ABB RAPID module: P103.mod

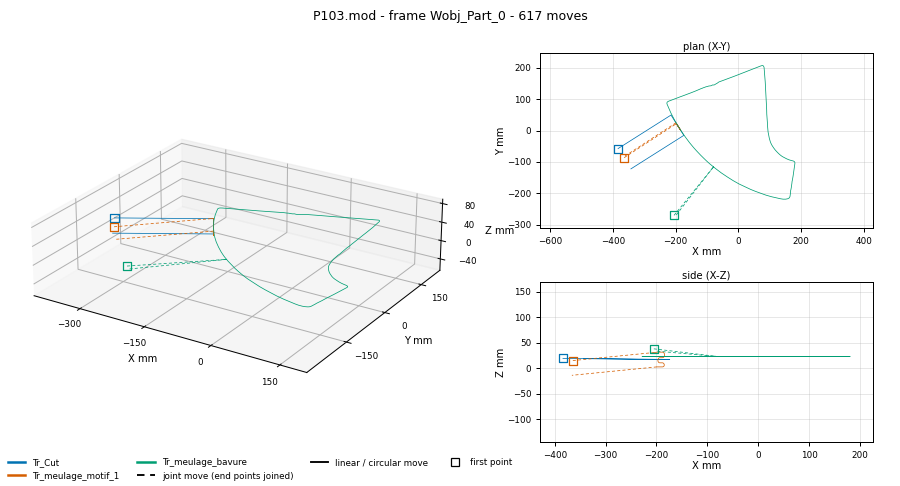
[picture p0: tool path of P103.mod in frame Wobj_Part_0, 617 of 625 moves have a stored position in this frame; points joined in program order, loops and branches not executed]
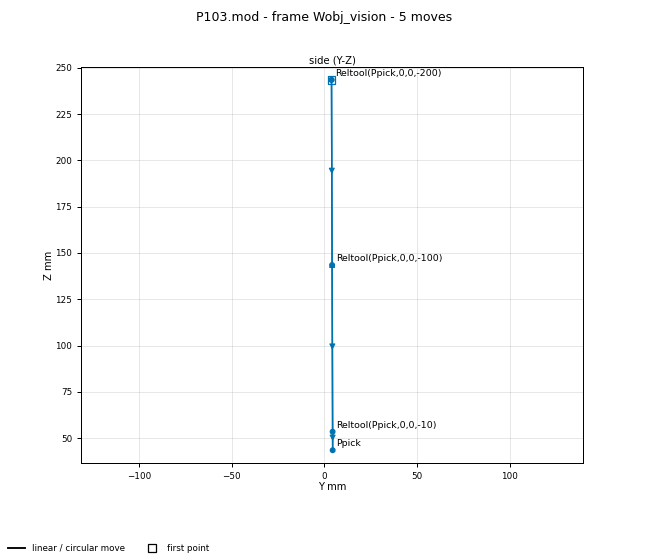
[picture p1: tool path of P103.mod in frame Wobj_vision, 5 of 625 moves have a stored position in this frame; points joined in program order, loops and branches not executed]
MODULE P103
	LOCAL CONST Speeddata vitesse_Tronconnage :=[10, 500, 0, 0];
	LOCAL CONST Robtarget Coupe_0 :=[[-191.77609375,12.892310546875,17.173708984375],[0.680249271326253,0.678001155670585,0.200784543502111,0.193030901308835],[0,0,0,0],[8.999999E+09,8.999999E+09,8.999999E+09,8.999999E+09,8.999999E+09,8.999999E+09]];
	LOCAL CONST Robtarget Tr_meulage_motif_1_App1 :=[[-364.480910820686,-86.5896332823026,15.1430730099713],[0.64692434542493,-0.59549439899172,0.32258675367408,-0.350446998018296],[0,0,0,0],[8.999999E+09,8.999999E+09,8.999999E+09,8.999999E+09,8.999999E+09,8.999999E+09]];
	LOCAL CONST Robtarget Tr_meulage_motif_1_App2 :=[[-205.877100228534,16.8426673593224,30.8462717169048],[0.64692434542493,-0.59549439899172,0.32258675367408,-0.350446998018296],[0,0,0,0],[8.999999E+09,8.999999E+09,8.999999E+09,8.999999E+09,8.999999E+09,8.999999E+09]];
	LOCAL CONST Robtarget Tr_meulage_motif_1_P0 :=[[-197.52953125,22.28647265625,31.672755859375],[0.64692434542493,-0.59549439899172,0.32258675367408,-0.350446998018296],[0,0,0,0],[8.999999E+09,8.999999E+09,8.999999E+09,8.999999E+09,8.999999E+09,8.999999E+09]];
	LOCAL CONST Robtarget Tr_meulage_motif_1_P1 :=[[-196.9945,21.441646484375,31.672755859375],[0.64692434542493,-0.59549439899172,0.32258675367408,-0.350446998018296],[0,0,0,0],[8.999999E+09,8.999999E+09,8.999999E+09,8.999999E+09,8.999999E+09,8.999999E+09]];
	LOCAL CONST Robtarget Tr_meulage_motif_1_P2 :=[[-196.459453125,20.5968203125,31.6727578125],[0.64692434542493,-0.59549439899172,0.32258675367408,-0.350446998018296],[0,0,0,0],[8.999999E+09,8.999999E+09,8.999999E+09,8.999999E+09,8.999999E+09,8.999999E+09]];
	LOCAL CONST Robtarget Tr_meulage_motif_1_P3 :=[[-195.92440625,19.75199609375,31.6727578125],[0.64692434542493,-0.59549439899172,0.32258675367408,-0.350446998018296],[0,0,0,0],[8.999999E+09,8.999999E+09,8.999999E+09,8.999999E+09,8.999999E+09,8.999999E+09]];
	LOCAL CONST Robtarget Tr_meulage_motif_1_P4 :=[[-195.389375,18.907169921875,31.6727578125],[0.64692434542493,-0.59549439899172,0.32258675367408,-0.350446998018296],[0,0,0,0],[8.999999E+09,8.999999E+09,8.999999E+09,8.999999E+09,8.999999E+09,8.999999E+09]];
	LOCAL CONST Robtarget Tr_meulage_motif_1_P5 :=[[-194.854328125,18.06234375,31.672759765625],[0.64692434542493,-0.59549439899172,0.32258675367408,-0.350446998018296],[0,0,0,0],[8.999999E+09,8.999999E+09,8.999999E+09,8.999999E+09,8.999999E+09,8.999999E+09]];
	LOCAL CONST Robtarget Tr_meulage_motif_1_P6 :=[[-194.31928125,17.217517578125,31.672759765625],[0.64692434542493,-0.59549439899172,0.32258675367408,-0.350446998018296],[0,0,0,0],[8.999999E+09,8.999999E+09,8.999999E+09,8.999999E+09,8.999999E+09,8.999999E+09]];
	LOCAL CONST Robtarget Tr_meulage_motif_1_P7 :=[[-193.78425,16.3726923828125,31.672759765625],[0.64692434542493,-0.59549439899172,0.32258675367408,-0.350446998018296],[0,0,0,0],[8.999999E+09,8.999999E+09,8.999999E+09,8.999999E+09,8.999999E+09,8.999999E+09]];
	LOCAL CONST Robtarget Tr_meulage_motif_1_P8 :=[[-193.249203125,15.5278671875,31.67276171875],[0.64692434542493,-0.59549439899172,0.32258675367408,-0.350446998018296],[0,0,0,0],[8.999999E+09,8.999999E+09,8.999999E+09,8.999999E+09,8.999999E+09,8.999999E+09]];
	LOCAL CONST Robtarget Tr_meulage_motif_1_P9 :=[[-192.71415625,14.683041015625,31.67276171875],[0.64692434542493,-0.59549439899172,0.32258675367408,-0.350446998018296],[0,0,0,0],[8.999999E+09,8.999999E+09,8.999999E+09,8.999999E+09,8.999999E+09,8.999999E+09]];
	LOCAL CONST Robtarget Tr_meulage_motif_1_P10 :=[[-192.179125,13.8382158203125,31.67276171875],[0.64692434542493,-0.59549439899172,0.32258675367408,-0.350446998018296],[0,0,0,0],[8.999999E+09,8.999999E+09,8.999999E+09,8.999999E+09,8.999999E+09,8.999999E+09]];
	LOCAL CONST Robtarget Tr_meulage_motif_1_P11 :=[[-191.644078125,12.9933896484375,31.672763671875],[0.64692434542493,-0.59549439899172,0.32258675367408,-0.350446998018296],[0,0,0,0],[8.999999E+09,8.999999E+09,8.999999E+09,8.999999E+09,8.999999E+09,8.999999E+09]];
	LOCAL CONST Robtarget Tr_meulage_motif_1_P12 :=[[-191.10903125,12.148564453125,31.672763671875],[0.64692434542493,-0.59549439899172,0.32258675367408,-0.350446998018296],[0,0,0,0],[8.999999E+09,8.999999E+09,8.999999E+09,8.999999E+09,8.999999E+09,8.999999E+09]];
	LOCAL CONST Robtarget Tr_meulage_motif_1_P13 :=[[-190.574,11.30373828125,31.672763671875],[0.64692434542493,-0.59549439899172,0.32258675367408,-0.350446998018296],[0,0,0,0],[8.999999E+09,8.999999E+09,8.999999E+09,8.999999E+09,8.999999E+09,8.999999E+09]];
	LOCAL CONST Robtarget Tr_meulage_motif_1_P14 :=[[-190.038953125,10.4589130859375,31.672765625],[0.64692434542493,-0.59549439899172,0.32258675367408,-0.350446998018296],[0,0,0,0],[8.999999E+09,8.999999E+09,8.999999E+09,8.999999E+09,8.999999E+09,8.999999E+09]];
	LOCAL CONST Robtarget Tr_meulage_motif_1_P15 :=[[-189.50390625,9.6140869140625,31.672765625],[0.64692434542493,-0.59549439899172,0.32258675367408,-0.350446998018296],[0,0,0,0],[8.999999E+09,8.999999E+09,8.999999E+09,8.999999E+09,8.999999E+09,8.999999E+09]];
	LOCAL CONST Robtarget Tr_meulage_motif_1_P16 :=[[-188.968875,8.76926171875,31.672765625],[0.64692434542493,-0.59549439899172,0.32258675367408,-0.350446998018296],[0,0,0,0],[8.999999E+09,8.999999E+09,8.999999E+09,8.999999E+09,8.999999E+09,8.999999E+09]];
	LOCAL CONST Robtarget Tr_meulage_motif_1_P17 :=[[-188.433828125,7.92443603515625,31.672767578125],[0.64692434542493,-0.59549439899172,0.32258675367408,-0.350446998018296],[0,0,0,0],[8.999999E+09,8.999999E+09,8.999999E+09,8.999999E+09,8.999999E+09,8.999999E+09]];
	LOCAL CONST Robtarget Tr_meulage_motif_1_P18 :=[[-187.89878125,7.0796103515625,31.672767578125],[0.64692434542493,-0.59549439899172,0.32258675367408,-0.350446998018296],[0,0,0,0],[8.999999E+09,8.999999E+09,8.999999E+09,8.999999E+09,8.999999E+09,8.999999E+09]];
	LOCAL CONST Robtarget Tr_meulage_motif_1_P19 :=[[-187.368796875,6.24039208984375,31.562181640625],[0.64692434542493,-0.59549439899172,0.32258675367408,-0.350446998018296],[0,0,0,0],[8.999999E+09,8.999999E+09,8.999999E+09,8.999999E+09,8.999999E+09,8.999999E+09]];
	LOCAL CONST Robtarget Tr_meulage_motif_1_P20 :=[[-186.86440625,5.4394736328125,31.351009765625],[0.64692434542493,-0.59549439899172,0.32258675367408,-0.350446998018296],[0,0,0,0],[8.999999E+09,8.999999E+09,8.999999E+09,8.999999E+09,8.999999E+09,8.999999E+09]];
	LOCAL CONST Robtarget Tr_meulage_motif_1_P21 :=[[-186.410796875,4.71741357421875,31.07918359375],[0.64692434542493,-0.59549439899172,0.32258675367408,-0.350446998018296],[0,0,0,0],[8.999999E+09,8.999999E+09,8.999999E+09,8.999999E+09,8.999999E+09,8.999999E+09]];
	LOCAL CONST Robtarget Tr_meulage_motif_1_P22 :=[[-186.012203125,4.08216088867187,30.803263671875],[0.64692434542493,-0.59549439899172,0.32258675367408,-0.350446998018296],[0,0,0,0],[8.999999E+09,8.999999E+09,8.999999E+09,8.999999E+09,8.999999E+09,8.999999E+09]];
	LOCAL CONST Robtarget Tr_meulage_motif_1_P23 :=[[-185.42903125,3.148189453125,30.1871796875],[0.64692434542493,-0.59549439899172,0.32258675367408,-0.350446998018296],[0,0,0,0],[8.999999E+09,8.999999E+09,8.999999E+09,8.999999E+09,8.999999E+09,8.999999E+09]];
	LOCAL CONST Robtarget Tr_meulage_motif_1_P24 :=[[-184.88940625,2.27801293945312,29.339580078125],[0.64692434542493,-0.59549439899172,0.32258675367408,-0.350446998018296],[0,0,0,0],[8.999999E+09,8.999999E+09,8.999999E+09,8.999999E+09,8.999999E+09,8.999999E+09]];
	LOCAL CONST Robtarget Tr_meulage_motif_1_P25 :=[[-184.44575,1.55563366699219,28.315771484375],[0.64692434542493,-0.59549439899172,0.32258675367408,-0.350446998018296],[0,0,0,0],[8.999999E+09,8.999999E+09,8.999999E+09,8.999999E+09,8.999999E+09,8.999999E+09]];
	LOCAL CONST Robtarget Tr_meulage_motif_1_P26 :=[[-184.195328125,1.13640502929688,27.199658203125],[0.64692434542493,-0.59549439899172,0.32258675367408,-0.350446998018296],[0,0,0,0],[8.999999E+09,8.999999E+09,8.999999E+09,8.999999E+09,8.999999E+09,8.999999E+09]];
	LOCAL CONST Robtarget Tr_meulage_motif_1_P27 :=[[-184.187578125,1.10928845214844,26.503734375],[0.64692434542493,-0.59549439899172,0.32258675367408,-0.350446998018296],[0,0,0,0],[8.999999E+09,8.999999E+09,8.999999E+09,8.999999E+09,8.999999E+09,8.999999E+09]];
	LOCAL CONST Robtarget Tr_meulage_motif_1_P28 :=[[-184.193953125,1.10524719238281,25.84252734375],[0.64692434542493,-0.59549439899172,0.32258675367408,-0.350446998018296],[0,0,0,0],[8.999999E+09,8.999999E+09,8.999999E+09,8.999999E+09,8.999999E+09,8.999999E+09]];
	LOCAL CONST Robtarget Tr_meulage_motif_1_P29 :=[[-184.2296875,1.14756665039062,25.1814765625],[0.64692434542493,-0.59549439899172,0.32258675367408,-0.350446998018296],[0,0,0,0],[8.999999E+09,8.999999E+09,8.999999E+09,8.999999E+09,8.999999E+09,8.999999E+09]];
	LOCAL CONST Robtarget Tr_meulage_motif_1_P30 :=[[-184.506890625,1.5617412109375,24.079798828125],[0.64692434542493,-0.59549439899172,0.32258675367408,-0.350446998018296],[0,0,0,0],[8.999999E+09,8.999999E+09,8.999999E+09,8.999999E+09,8.999999E+09,8.999999E+09]];
	LOCAL CONST Robtarget Tr_meulage_motif_1_P31 :=[[-184.9749375,2.27928784179687,23.07323828125],[0.64692434542493,-0.59549439899172,0.32258675367408,-0.350446998018296],[0,0,0,0],[8.999999E+09,8.999999E+09,8.999999E+09,8.999999E+09,8.999999E+09,8.999999E+09]];
	LOCAL CONST Robtarget Tr_meulage_motif_1_P32 :=[[-185.5305,3.13882202148437,22.24441796875],[0.64692434542493,-0.59549439899172,0.32258675367408,-0.350446998018296],[0,0,0,0],[8.999999E+09,8.999999E+09,8.999999E+09,8.999999E+09,8.999999E+09,8.999999E+09]];
	LOCAL CONST Robtarget Tr_meulage_motif_1_P33 :=[[-185.9019375,3.71687768554688,21.848693359375],[0.64692434542493,-0.59549439899172,0.32258675367408,-0.350446998018296],[0,0,0,0],[8.999999E+09,8.999999E+09,8.999999E+09,8.999999E+09,8.999999E+09,8.999999E+09]];
	LOCAL CONST Robtarget Tr_meulage_motif_1_P34 :=[[-186.526296875,4.69233837890625,21.36119140625],[0.64692434542493,-0.59549439899172,0.32258675367408,-0.350446998018296],[0,0,0,0],[8.999999E+09,8.999999E+09,8.999999E+09,8.999999E+09,8.999999E+09,8.999999E+09]];
	LOCAL CONST Robtarget Tr_meulage_motif_1_P35 :=[[-186.980984375,5.40462841796875,21.097115234375],[0.64692434542493,-0.59549439899172,0.32258675367408,-0.350446998018296],[0,0,0,0],[8.999999E+09,8.999999E+09,8.999999E+09,8.999999E+09,8.999999E+09,8.999999E+09]];
	LOCAL CONST Robtarget Tr_meulage_motif_1_P36 :=[[-187.481609375,6.19075634765625,20.89266015625],[0.64692434542493,-0.59549439899172,0.32258675367408,-0.350446998018296],[0,0,0,0],[8.999999E+09,8.999999E+09,8.999999E+09,8.999999E+09,8.999999E+09,8.999999E+09]];
	LOCAL CONST Robtarget Tr_meulage_motif_1_P37 :=[[-188.007828125,7.019341796875,20.784072265625],[0.64692434542493,-0.59549439899172,0.32258675367408,-0.350446998018296],[0,0,0,0],[8.999999E+09,8.999999E+09,8.999999E+09,8.999999E+09,8.999999E+09,8.999999E+09]];
	LOCAL CONST Robtarget Tr_meulage_motif_1_P38 :=[[-188.53996875,7.8572080078125,20.673484375],[0.64692434542493,-0.59549439899172,0.32258675367408,-0.350446998018296],[0,0,0,0],[8.999999E+09,8.999999E+09,8.999999E+09,8.999999E+09,8.999999E+09,8.999999E+09]];
	LOCAL CONST Robtarget Tr_meulage_motif_1_P39 :=[[-189.075,8.7020341796875,20.673484375],[0.64692434542493,-0.59549439899172,0.32258675367408,-0.350446998018296],[0,0,0,0],[8.999999E+09,8.999999E+09,8.999999E+09,8.999999E+09,8.999999E+09,8.999999E+09]];
	LOCAL CONST Robtarget Tr_meulage_motif_1_P40 :=[[-189.610046875,9.546859375,20.673482421875],[0.64692434542493,-0.59549439899172,0.32258675367408,-0.350446998018296],[0,0,0,0],[8.999999E+09,8.999999E+09,8.999999E+09,8.999999E+09,8.999999E+09,8.999999E+09]];
	LOCAL CONST Robtarget Tr_meulage_motif_1_P41 :=[[-190.14509375,10.391685546875,20.673482421875],[0.64692434542493,-0.59549439899172,0.32258675367408,-0.350446998018296],[0,0,0,0],[8.999999E+09,8.999999E+09,8.999999E+09,8.999999E+09,8.999999E+09,8.999999E+09]];
	LOCAL CONST Robtarget Tr_meulage_motif_1_P42 :=[[-190.680125,11.2365107421875,20.673482421875],[0.64692434542493,-0.59549439899172,0.32258675367408,-0.350446998018296],[0,0,0,0],[8.999999E+09,8.999999E+09,8.999999E+09,8.999999E+09,8.999999E+09,8.999999E+09]];
	LOCAL CONST Robtarget Tr_meulage_motif_1_P43 :=[[-191.215171875,12.0813369140625,20.67348046875],[0.64692434542493,-0.59549439899172,0.32258675367408,-0.350446998018296],[0,0,0,0],[8.999999E+09,8.999999E+09,8.999999E+09,8.999999E+09,8.999999E+09,8.999999E+09]];
	LOCAL CONST Robtarget Tr_meulage_motif_1_P44 :=[[-191.75021875,12.926162109375,20.67348046875],[0.64692434542493,-0.59549439899172,0.32258675367408,-0.350446998018296],[0,0,0,0],[8.999999E+09,8.999999E+09,8.999999E+09,8.999999E+09,8.999999E+09,8.999999E+09]];
	LOCAL CONST Robtarget Tr_meulage_motif_1_P45 :=[[-192.28525,13.77098828125,20.67348046875],[0.64692434542493,-0.59549439899172,0.32258675367408,-0.350446998018296],[0,0,0,0],[8.999999E+09,8.999999E+09,8.999999E+09,8.999999E+09,8.999999E+09,8.999999E+09]];
	LOCAL CONST Robtarget Tr_meulage_motif_1_P46 :=[[-192.820296875,14.6158134765625,20.673478515625],[0.64692434542493,-0.59549439899172,0.32258675367408,-0.350446998018296],[0,0,0,0],[8.999999E+09,8.999999E+09,8.999999E+09,8.999999E+09,8.999999E+09,8.999999E+09]];
	LOCAL CONST Robtarget Tr_meulage_motif_1_P47 :=[[-193.35534375,15.4606396484375,20.673478515625],[0.64692434542493,-0.59549439899172,0.32258675367408,-0.350446998018296],[0,0,0,0],[8.999999E+09,8.999999E+09,8.999999E+09,8.999999E+09,8.999999E+09,8.999999E+09]];
	LOCAL CONST Robtarget Tr_meulage_motif_1_P48 :=[[-193.890375,16.30546484375,20.673478515625],[0.64692434542493,-0.59549439899172,0.32258675367408,-0.350446998018296],[0,0,0,0],[8.999999E+09,8.999999E+09,8.999999E+09,8.999999E+09,8.999999E+09,8.999999E+09]];
	LOCAL CONST Robtarget Tr_meulage_motif_1_P49 :=[[-194.422515625,17.14333203125,20.562890625],[0.64692434542493,-0.59549439899172,0.32258675367408,-0.350446998018296],[0,0,0,0],[8.999999E+09,8.999999E+09,8.999999E+09,8.999999E+09,8.999999E+09,8.999999E+09]];
	LOCAL CONST Robtarget Tr_meulage_motif_1_P50 :=[[-194.93096875,17.94166796875,20.351716796875],[0.64692434542493,-0.59549439899172,0.32258675367408,-0.350446998018296],[0,0,0,0],[8.999999E+09,8.999999E+09,8.999999E+09,8.999999E+09,8.999999E+09,8.999999E+09]];
	LOCAL CONST Robtarget Tr_meulage_motif_1_P51 :=[[-195.389828125,18.66040625,20.079890625],[0.64692434542493,-0.59549439899172,0.32258675367408,-0.350446998018296],[0,0,0,0],[8.999999E+09,8.999999E+09,8.999999E+09,8.999999E+09,8.999999E+09,8.999999E+09]];
	LOCAL CONST Robtarget Tr_meulage_motif_1_P52 :=[[-195.7734375,19.259640625,19.77575390625],[0.64692434542493,-0.59549439899172,0.32258675367408,-0.350446998018296],[0,0,0,0],[8.999999E+09,8.999999E+09,8.999999E+09,8.999999E+09,8.999999E+09,8.999999E+09]];
	LOCAL CONST Robtarget Tr_meulage_motif_1_P53 :=[[-196.333328125,20.129537109375,19.113263671875],[0.64692434542493,-0.59549439899172,0.32258675367408,-0.350446998018296],[0,0,0,0],[8.999999E+09,8.999999E+09,8.999999E+09,8.999999E+09,8.999999E+09,8.999999E+09]];
	LOCAL CONST Robtarget Tr_meulage_motif_1_P54 :=[[-196.82459375,20.88600390625,18.211384765625],[0.64692434542493,-0.59549439899172,0.32258675367408,-0.350446998018296],[0,0,0,0],[8.999999E+09,8.999999E+09,8.999999E+09,8.999999E+09,8.999999E+09,8.999999E+09]];
	LOCAL CONST Robtarget Tr_meulage_motif_1_P55 :=[[-197.120921875,21.33156640625,17.165421875],[0.64692434542493,-0.59549439899172,0.32258675367408,-0.350446998018296],[0,0,0,0],[8.999999E+09,8.999999E+09,8.999999E+09,8.999999E+09,8.999999E+09,8.999999E+09]];
	LOCAL CONST Robtarget Tr_meulage_motif_1_P56 :=[[-197.22646875,21.4834375,16.472248046875],[0.64692434542493,-0.59549439899172,0.32258675367408,-0.350446998018296],[0,0,0,0],[8.999999E+09,8.999999E+09,8.999999E+09,8.999999E+09,8.999999E+09,8.999999E+09]];
	LOCAL CONST Robtarget Tr_meulage_motif_1_P57 :=[[-197.2680625,21.532669921875,15.7022978515625],[0.64692434542493,-0.59549439899172,0.32258675367408,-0.350446998018296],[0,0,0,0],[8.999999E+09,8.999999E+09,8.999999E+09,8.999999E+09,8.999999E+09,8.999999E+09]];
	LOCAL CONST Robtarget Tr_meulage_motif_1_P58 :=[[-197.239671875,21.4714140625,14.9324736328125],[0.64692434542493,-0.59549439899172,0.32258675367408,-0.350446998018296],[0,0,0,0],[8.999999E+09,8.999999E+09,8.999999E+09,8.999999E+09,8.999999E+09,8.999999E+09]];
	LOCAL CONST Robtarget Tr_meulage_motif_1_P59 :=[[-197.025875,21.11015625,13.8242958984375],[0.64692434542493,-0.59549439899172,0.32258675367408,-0.350446998018296],[0,0,0,0],[8.999999E+09,8.999999E+09,8.999999E+09,8.999999E+09,8.999999E+09,8.999999E+09]];
	LOCAL CONST Robtarget Tr_meulage_motif_1_P60 :=[[-196.80984375,20.7565546875,13.238646484375],[0.64692434542493,-0.59549439899172,0.32258675367408,-0.350446998018296],[0,0,0,0],[8.999999E+09,8.999999E+09,8.999999E+09,8.999999E+09,8.999999E+09,8.999999E+09]];
	LOCAL CONST Robtarget Tr_meulage_motif_1_P61 :=[[-196.343765625,20.00166796875,12.351580078125],[0.64692434542493,-0.59549439899172,0.32258675367408,-0.350446998018296],[0,0,0,0],[8.999999E+09,8.999999E+09,8.999999E+09,8.999999E+09,8.999999E+09,8.999999E+09]];
	LOCAL CONST Robtarget Tr_meulage_motif_1_P62 :=[[-196.034390625,19.50433203125,11.937294921875],[0.64692434542493,-0.59549439899172,0.32258675367408,-0.350446998018296],[0,0,0,0],[8.999999E+09,8.999999E+09,8.999999E+09,8.999999E+09,8.999999E+09,8.999999E+09]];
	LOCAL CONST Robtarget Tr_meulage_motif_1_P63 :=[[-195.441515625,18.5565703125,11.39323828125],[0.64692434542493,-0.59549439899172,0.32258675367408,-0.350446998018296],[0,0,0,0],[8.999999E+09,8.999999E+09,8.999999E+09,8.999999E+09,8.999999E+09,8.999999E+09]];
	LOCAL CONST Robtarget Tr_meulage_motif_1_P64 :=[[-195.002640625,17.85728125,11.0977578125],[0.64692434542493,-0.59549439899172,0.32258675367408,-0.350446998018296],[0,0,0,0],[8.999999E+09,8.999999E+09,8.999999E+09,8.999999E+09,8.999999E+09,8.999999E+09]];
	LOCAL CONST Robtarget Tr_meulage_motif_1_P65 :=[[-194.505953125,17.068654296875,10.893302734375],[0.64692434542493,-0.59549439899172,0.32258675367408,-0.350446998018296],[0,0,0,0],[8.999999E+09,8.999999E+09,8.999999E+09,8.999999E+09,8.999999E+09,8.999999E+09]];
	LOCAL CONST Robtarget Tr_meulage_motif_1_P66 :=[[-193.981828125,16.2387412109375,10.784716796875],[0.64692434542493,-0.59549439899172,0.32258675367408,-0.350446998018296],[0,0,0,0],[8.999999E+09,8.999999E+09,8.999999E+09,8.999999E+09,8.999999E+09,8.999999E+09]];
	LOCAL CONST Robtarget Tr_meulage_motif_1_P67 :=[[-193.451828125,15.3995234375,10.674130859375],[0.64692434542493,-0.59549439899172,0.32258675367408,-0.350446998018296],[0,0,0,0],[8.999999E+09,8.999999E+09,8.999999E+09,8.999999E+09,8.999999E+09,8.999999E+09]];
	LOCAL CONST Robtarget Tr_meulage_motif_1_P68 :=[[-192.91678125,14.554697265625,10.6741318359375],[0.64692434542493,-0.59549439899172,0.32258675367408,-0.350446998018296],[0,0,0,0],[8.999999E+09,8.999999E+09,8.999999E+09,8.999999E+09,8.999999E+09,8.999999E+09]];
	LOCAL CONST Robtarget Tr_meulage_motif_1_P69 :=[[-192.38175,13.7098720703125,10.6741318359375],[0.64692434542493,-0.59549439899172,0.32258675367408,-0.350446998018296],[0,0,0,0],[8.999999E+09,8.999999E+09,8.999999E+09,8.999999E+09,8.999999E+09,8.999999E+09]];
	LOCAL CONST Robtarget Tr_meulage_motif_1_P70 :=[[-191.846703125,12.8650458984375,10.6741328125],[0.64692434542493,-0.59549439899172,0.32258675367408,-0.350446998018296],[0,0,0,0],[8.999999E+09,8.999999E+09,8.999999E+09,8.999999E+09,8.999999E+09,8.999999E+09]];
	LOCAL CONST Robtarget Tr_meulage_motif_1_P71 :=[[-191.31165625,12.020220703125,10.6741337890625],[0.64692434542493,-0.59549439899172,0.32258675367408,-0.350446998018296],[0,0,0,0],[8.999999E+09,8.999999E+09,8.999999E+09,8.999999E+09,8.999999E+09,8.999999E+09]];
	LOCAL CONST Robtarget Tr_meulage_motif_1_P72 :=[[-190.776625,11.17539453125,10.674134765625],[0.64692434542493,-0.59549439899172,0.32258675367408,-0.350446998018296],[0,0,0,0],[8.999999E+09,8.999999E+09,8.999999E+09,8.999999E+09,8.999999E+09,8.999999E+09]];
	LOCAL CONST Robtarget Tr_meulage_motif_1_P73 :=[[-190.241578125,10.3305693359375,10.674134765625],[0.64692434542493,-0.59549439899172,0.32258675367408,-0.350446998018296],[0,0,0,0],[8.999999E+09,8.999999E+09,8.999999E+09,8.999999E+09,8.999999E+09,8.999999E+09]];
	LOCAL CONST Robtarget Tr_meulage_motif_1_P74 :=[[-189.70653125,9.4857431640625,10.6741357421875],[0.64692434542493,-0.59549439899172,0.32258675367408,-0.350446998018296],[0,0,0,0],[8.999999E+09,8.999999E+09,8.999999E+09,8.999999E+09,8.999999E+09,8.999999E+09]];
	LOCAL CONST Robtarget Tr_meulage_motif_1_P75 :=[[-189.1715,8.64091796875,10.67413671875],[0.64692434542493,-0.59549439899172,0.32258675367408,-0.350446998018296],[0,0,0,0],[8.999999E+09,8.999999E+09,8.999999E+09,8.999999E+09,8.999999E+09,8.999999E+09]];
	LOCAL CONST Robtarget Tr_meulage_motif_1_P76 :=[[-188.636453125,7.79609228515625,10.67413671875],[0.64692434542493,-0.59549439899172,0.32258675367408,-0.350446998018296],[0,0,0,0],[8.999999E+09,8.999999E+09,8.999999E+09,8.999999E+09,8.999999E+09,8.999999E+09]];
	LOCAL CONST Robtarget Tr_meulage_motif_1_P77 :=[[-188.10140625,6.9512666015625,10.6741376953125],[0.64692434542493,-0.59549439899172,0.32258675367408,-0.350446998018296],[0,0,0,0],[8.999999E+09,8.999999E+09,8.999999E+09,8.999999E+09,8.999999E+09,8.999999E+09]];
	LOCAL CONST Robtarget Tr_meulage_motif_1_P78 :=[[-187.571421875,6.11204833984375,10.5635517578125],[0.64692434542493,-0.59549439899172,0.32258675367408,-0.350446998018296],[0,0,0,0],[8.999999E+09,8.999999E+09,8.999999E+09,8.999999E+09,8.999999E+09,8.999999E+09]];
	LOCAL CONST Robtarget Tr_meulage_motif_1_P79 :=[[-187.06703125,5.31113037109375,10.35237890625],[0.64692434542493,-0.59549439899172,0.32258675367408,-0.350446998018296],[0,0,0,0],[8.999999E+09,8.999999E+09,8.999999E+09,8.999999E+09,8.999999E+09,8.999999E+09]];
	LOCAL CONST Robtarget Tr_meulage_motif_1_P80 :=[[-186.613421875,4.58906982421875,10.080552734375],[0.64692434542493,-0.59549439899172,0.32258675367408,-0.350446998018296],[0,0,0,0],[8.999999E+09,8.999999E+09,8.999999E+09,8.999999E+09,8.999999E+09,8.999999E+09]];
	LOCAL CONST Robtarget Tr_meulage_motif_1_P81 :=[[-186.214828125,3.95381713867188,9.8046337890625],[0.64692434542493,-0.59549439899172,0.32258675367408,-0.350446998018296],[0,0,0,0],[8.999999E+09,8.999999E+09,8.999999E+09,8.999999E+09,8.999999E+09,8.999999E+09]];
	LOCAL CONST Robtarget Tr_meulage_motif_1_P82 :=[[-185.631671875,3.019845703125,9.1885498046875],[0.64692434542493,-0.59549439899172,0.32258675367408,-0.350446998018296],[0,0,0,0],[8.999999E+09,8.999999E+09,8.999999E+09,8.999999E+09,8.999999E+09,8.999999E+09]];
	LOCAL CONST Robtarget Tr_meulage_motif_1_P83 :=[[-185.12840625,2.20612158203125,8.294640625],[0.64692434542493,-0.59549439899172,0.32258675367408,-0.350446998018296],[0,0,0,0],[8.999999E+09,8.999999E+09,8.999999E+09,8.999999E+09,8.999999E+09,8.999999E+09]];
	LOCAL CONST Robtarget Tr_meulage_motif_1_P84 :=[[-184.812984375,1.68488000488281,7.20871142578125],[0.64692434542493,-0.59549439899172,0.32258675367408,-0.350446998018296],[0,0,0,0],[8.999999E+09,8.999999E+09,8.999999E+09,8.999999E+09,8.999999E+09,8.999999E+09]];
	LOCAL CONST Robtarget Tr_meulage_motif_1_P85 :=[[-184.731890625,1.53582434082031,6.22440087890625],[0.64692434542493,-0.59549439899172,0.32258675367408,-0.350446998018296],[0,0,0,0],[8.999999E+09,8.999999E+09,8.999999E+09,8.999999E+09,8.999999E+09,8.999999E+09]];
	LOCAL CONST Robtarget Tr_meulage_motif_1_P86 :=[[-184.804203125,1.64564172363281,6.0197578125],[0.64692434542493,-0.59549439899172,0.32258675367408,-0.350446998018296],[0,0,0,0],[8.999999E+09,8.999999E+09,8.999999E+09,8.999999E+09,8.999999E+09,8.999999E+09]];
	LOCAL CONST Robtarget Tr_meulage_motif_1_P87 :=[[-184.87721875,1.7454326171875,5.29339892578125],[0.64692434542493,-0.59549439899172,0.32258675367408,-0.350446998018296],[0,0,0,0],[8.999999E+09,8.999999E+09,8.999999E+09,8.999999E+09,8.999999E+09,8.999999E+09]];
	LOCAL CONST Robtarget Tr_meulage_motif_1_P88 :=[[-185.252234375,2.3175673828125,4.35655322265625],[0.64692434542493,-0.59549439899172,0.32258675367408,-0.350446998018296],[0,0,0,0],[8.999999E+09,8.999999E+09,8.999999E+09,8.999999E+09,8.999999E+09,8.999999E+09]];
	LOCAL CONST Robtarget Tr_meulage_motif_1_P89 :=[[-185.5550625,2.78582861328125,3.89277075195313],[0.64692434542493,-0.59549439899172,0.32258675367408,-0.350446998018296],[0,0,0,0],[8.999999E+09,8.999999E+09,8.999999E+09,8.999999E+09,8.999999E+09,8.999999E+09]];
	LOCAL CONST Robtarget Tr_meulage_motif_1_P90 :=[[-186.1649375,3.73750390625,3.3623671875],[0.64692434542493,-0.59549439899172,0.32258675367408,-0.350446998018296],[0,0,0,0],[8.999999E+09,8.999999E+09,8.999999E+09,8.999999E+09,8.999999E+09,8.999999E+09]];
	LOCAL CONST Robtarget Tr_meulage_motif_1_P91 :=[[-186.619625,4.4497939453125,3.0982900390625],[0.64692434542493,-0.59549439899172,0.32258675367408,-0.350446998018296],[0,0,0,0],[8.999999E+09,8.999999E+09,8.999999E+09,8.999999E+09,8.999999E+09,8.999999E+09]];
	LOCAL CONST Robtarget Tr_meulage_motif_1_P92 :=[[-187.12025,5.235921875,2.893833984375],[0.64692434542493,-0.59549439899172,0.32258675367408,-0.350446998018296],[0,0,0,0],[8.999999E+09,8.999999E+09,8.999999E+09,8.999999E+09,8.999999E+09,8.999999E+09]];
	LOCAL CONST Robtarget Tr_meulage_motif_1_P93 :=[[-187.64646875,6.06450732421875,2.78524658203125],[0.64692434542493,-0.59549439899172,0.32258675367408,-0.350446998018296],[0,0,0,0],[8.999999E+09,8.999999E+09,8.999999E+09,8.999999E+09,8.999999E+09,8.999999E+09]];
	LOCAL CONST Robtarget Tr_meulage_motif_1_P94 :=[[-188.178609375,6.90237353515625,2.67465942382813],[0.64692434542493,-0.59549439899172,0.32258675367408,-0.350446998018296],[0,0,0,0],[8.999999E+09,8.999999E+09,8.999999E+09,8.999999E+09,8.999999E+09,8.999999E+09]];
	LOCAL CONST Robtarget Tr_meulage_motif_1_P95 :=[[-188.713640625,7.74719921875,2.67465869140625],[0.64692434542493,-0.59549439899172,0.32258675367408,-0.350446998018296],[0,0,0,0],[8.999999E+09,8.999999E+09,8.999999E+09,8.999999E+09,8.999999E+09,8.999999E+09]];
	LOCAL CONST Robtarget Tr_meulage_motif_1_P96 :=[[-189.2486875,8.592025390625,2.674658203125],[0.64692434542493,-0.59549439899172,0.32258675367408,-0.350446998018296],[0,0,0,0],[8.999999E+09,8.999999E+09,8.999999E+09,8.999999E+09,8.999999E+09,8.999999E+09]];
	LOCAL CONST Robtarget Tr_meulage_motif_1_P97 :=[[-189.783734375,9.4368505859375,2.67465747070313],[0.64692434542493,-0.59549439899172,0.32258675367408,-0.350446998018296],[0,0,0,0],[8.999999E+09,8.999999E+09,8.999999E+09,8.999999E+09,8.999999E+09,8.999999E+09]];
	LOCAL CONST Robtarget Tr_meulage_motif_1_P98 :=[[-190.318765625,10.2816767578125,2.67465673828125],[0.64692434542493,-0.59549439899172,0.32258675367408,-0.350446998018296],[0,0,0,0],[8.999999E+09,8.999999E+09,8.999999E+09,8.999999E+09,8.999999E+09,8.999999E+09]];
	LOCAL CONST Robtarget Tr_meulage_motif_1_P99 :=[[-190.8538125,11.126501953125,2.67465600585937],[0.64692434542493,-0.59549439899172,0.32258675367408,-0.350446998018296],[0,0,0,0],[8.999999E+09,8.999999E+09,8.999999E+09,8.999999E+09,8.999999E+09,8.999999E+09]];
	LOCAL CONST Robtarget Tr_meulage_motif_1_P100 :=[[-191.388859375,11.971328125,2.67465551757813],[0.64692434542493,-0.59549439899172,0.32258675367408,-0.350446998018296],[0,0,0,0],[8.999999E+09,8.999999E+09,8.999999E+09,8.999999E+09,8.999999E+09,8.999999E+09]];
	LOCAL CONST Robtarget Tr_meulage_motif_1_P101 :=[[-191.923890625,12.8161533203125,2.67465478515625],[0.64692434542493,-0.59549439899172,0.32258675367408,-0.350446998018296],[0,0,0,0],[8.999999E+09,8.999999E+09,8.999999E+09,8.999999E+09,8.999999E+09,8.999999E+09]];
	LOCAL CONST Robtarget Tr_meulage_motif_1_P102 :=[[-192.4589375,13.6609794921875,2.67465405273437],[0.64692434542493,-0.59549439899172,0.32258675367408,-0.350446998018296],[0,0,0,0],[8.999999E+09,8.999999E+09,8.999999E+09,8.999999E+09,8.999999E+09,8.999999E+09]];
	LOCAL CONST Robtarget Tr_meulage_motif_1_P103 :=[[-192.993984375,14.5058046875,2.67465356445312],[0.64692434542493,-0.59549439899172,0.32258675367408,-0.350446998018296],[0,0,0,0],[8.999999E+09,8.999999E+09,8.999999E+09,8.999999E+09,8.999999E+09,8.999999E+09]];
	LOCAL CONST Robtarget Tr_meulage_motif_1_P104 :=[[-193.529015625,15.350630859375,2.67465283203125],[0.64692434542493,-0.59549439899172,0.32258675367408,-0.350446998018296],[0,0,0,0],[8.999999E+09,8.999999E+09,8.999999E+09,8.999999E+09,8.999999E+09,8.999999E+09]];
	LOCAL CONST Robtarget Tr_meulage_motif_1_P105 :=[[-194.0640625,16.1954560546875,2.67465209960938],[0.64692434542493,-0.59549439899172,0.32258675367408,-0.350446998018296],[0,0,0,0],[8.999999E+09,8.999999E+09,8.999999E+09,8.999999E+09,8.999999E+09,8.999999E+09]];
	LOCAL CONST Robtarget Tr_meulage_motif_1_P106 :=[[-194.599109375,17.04028125,2.6746513671875],[0.64692434542493,-0.59549439899172,0.32258675367408,-0.350446998018296],[0,0,0,0],[8.999999E+09,8.999999E+09,8.999999E+09,8.999999E+09,8.999999E+09,8.999999E+09]];
	LOCAL CONST Robtarget Tr_meulage_motif_1_P107 :=[[-195.134140625,17.885107421875,2.67465087890625],[0.64692434542493,-0.59549439899172,0.32258675367408,-0.350446998018296],[0,0,0,0],[8.999999E+09,8.999999E+09,8.999999E+09,8.999999E+09,8.999999E+09,8.999999E+09]];
	LOCAL CONST Robtarget Tr_meulage_motif_1_P108 :=[[-195.6691875,18.72993359375,2.67465014648438],[0.64692434542493,-0.59549439899172,0.32258675367408,-0.350446998018296],[0,0,0,0],[8.999999E+09,8.999999E+09,8.999999E+09,8.999999E+09,8.999999E+09,8.999999E+09]];
	LOCAL CONST Robtarget Tr_meulage_motif_1_P109 :=[[-196.204234375,19.574759765625,2.6746494140625],[0.64692434542493,-0.59549439899172,0.32258675367408,-0.350446998018296],[0,0,0,0],[8.999999E+09,8.999999E+09,8.999999E+09,8.999999E+09,8.999999E+09,8.999999E+09]];
	LOCAL CONST Robtarget Tr_meulage_motif_1_P110 :=[[-196.739265625,20.419583984375,2.67464868164063],[0.64692434542493,-0.59549439899172,0.32258675367408,-0.350446998018296],[0,0,0,0],[8.999999E+09,8.999999E+09,8.999999E+09,8.999999E+09,8.999999E+09,8.999999E+09]];
	LOCAL CONST Robtarget Tr_meulage_motif_1_P111 :=[[-197.2743125,21.26441015625,2.67464819335938],[0.64692434542493,-0.59549439899172,0.32258675367408,-0.350446998018296],[0,0,0,0],[8.999999E+09,8.999999E+09,8.999999E+09,8.999999E+09,8.999999E+09,8.999999E+09]];
	LOCAL CONST Robtarget Tr_meulage_motif_1_P112 :=[[-197.809359375,22.109236328125,2.6746474609375],[0.64692434542493,-0.59549439899172,0.32258675367408,-0.350446998018296],[0,0,0,0],[8.999999E+09,8.999999E+09,8.999999E+09,8.999999E+09,8.999999E+09,8.999999E+09]];
	LOCAL CONST Robtarget Tr_meulage_motif_1_P113 :=[[-198.344390625,22.9540625,2.67464672851563],[0.64692434542493,-0.59549439899172,0.32258675367408,-0.350446998018296],[0,0,0,0],[8.999999E+09,8.999999E+09,8.999999E+09,8.999999E+09,8.999999E+09,8.999999E+09]];
	LOCAL CONST Robtarget Tr_meulage_motif_1_P114 :=[[-198.8794375,23.79888671875,2.67464624023438],[0.64692434542493,-0.59549439899172,0.32258675367408,-0.350446998018296],[0,0,0,0],[8.999999E+09,8.999999E+09,8.999999E+09,8.999999E+09,8.999999E+09,8.999999E+09]];
	LOCAL CONST Robtarget Tr_meulage_motif_1_P115 :=[[-199.414484375,24.643712890625,2.6746455078125],[0.64692434542493,-0.59549439899172,0.32258675367408,-0.350446998018296],[0,0,0,0],[8.999999E+09,8.999999E+09,8.999999E+09,8.999999E+09,8.999999E+09,8.999999E+09]];
	LOCAL CONST Robtarget Tr_meulage_motif_1_degg1 :=[[-207.762053353534,19.1999075936974,1.84816136534232],[0.64692434542493,-0.59549439899172,0.32258675367408,-0.350446998018296],[0,0,0,0],[8.999999E+09,8.999999E+09,8.999999E+09,8.999999E+09,8.999999E+09,8.999999E+09]];
	LOCAL CONST Robtarget Tr_meulage_motif_1_degg2 :=[[-366.365863945686,-84.2323930479276,-13.8550373415912],[0.64692434542493,-0.59549439899172,0.32258675367408,-0.350446998018296],[0,0,0,0],[8.999999E+09,8.999999E+09,8.999999E+09,8.999999E+09,8.999999E+09,8.999999E+09]];
	LOCAL CONST Robtarget Tr_meulage_bavure_App1 :=[[-205.247085385378,-270.547663687165,38.1989633671395],[0.640389958710242,-0.691054659420384,0.245847241414717,-0.227822940823013],[0,0,0,0],[8.999999E+09,8.999999E+09,8.999999E+09,8.999999E+09,8.999999E+09,8.999999E+09]];
	LOCAL CONST Robtarget Tr_meulage_bavure_App2 :=[[-85.5941257536439,-123.664430840608,23.759948168357],[0.640389958710242,-0.691054659420384,0.245847241414717,-0.227822940823013],[0,0,0,0],[8.999999E+09,8.999999E+09,8.999999E+09,8.999999E+09,8.999999E+09,8.999999E+09]];
	LOCAL CONST Robtarget Tr_meulage_bavure_P0 :=[[-79.2966015625,-115.933734375,23],[0.640389958710242,-0.691054659420384,0.245847241414717,-0.227822940823013],[0,0,0,0],[8.999999E+09,8.999999E+09,8.999999E+09,8.999999E+09,8.999999E+09,8.999999E+09]];
	LOCAL CONST Robtarget Tr_meulage_bavure_P1 :=[[-85.8425,-110.82015625,23],[0.640277261040228,-0.690837470782079,0.246317331355744,-0.228290144842104],[0,0,0,0],[8.999999E+09,8.999999E+09,8.999999E+09,8.999999E+09,8.999999E+09,8.999999E+09]];
	LOCAL CONST Robtarget Tr_meulage_bavure_P2 :=[[-86.521640625,-110.2841484375,23],[0.639980724701222,-0.69020641145412,0.247628180674806,-0.229608505361214],[0,0,0,0],[8.999999E+09,8.999999E+09,8.999999E+09,8.999999E+09,8.999999E+09,8.999999E+09]];
	LOCAL CONST Robtarget Tr_meulage_bavure_P3 :=[[-86.9234296875,-109.95715625,23],[0.639566144574364,-0.689245369576477,0.249549287095217,-0.231562346986591],[0,0,0,0],[8.999999E+09,8.999999E+09,8.999999E+09,8.999999E+09,8.999999E+09,8.999999E+09]];
	LOCAL CONST Robtarget Tr_meulage_bavure_P4 :=[[-90.2432265625,-107.1154921875,23],[0.639117298896565,-0.688065539404016,0.251787655861441,-0.233875753535119],[0,0,0,0],[8.999999E+09,8.999999E+09,8.999999E+09,8.999999E+09,8.999999E+09,8.999999E+09]];
	LOCAL CONST Robtarget Tr_meulage_bavure_P5 :=[[-91.8843359375,-105.69653125,23],[0.63870801388743,-0.686759930540584,0.254098423436772,-0.2363194067503],[0,0,0,0],[8.999999E+09,8.999999E+09,8.999999E+09,8.999999E+09,8.999999E+09,8.999999E+09]];
	LOCAL CONST Robtarget Tr_meulage_bavure_P6 :=[[-91.9569375,-105.614515625,23],[0.638366793320061,-0.685382617078505,0.256365138021337,-0.238779022110784],[0,0,0,0],[8.999999E+09,8.999999E+09,8.999999E+09,8.999999E+09,8.999999E+09,8.999999E+09]];
	LOCAL CONST Robtarget Tr_meulage_bavure_P7 :=[[-93.0571015625,-104.660140625,23],[0.638080636724672,-0.683941529097321,0.258596686972375,-0.241256791199682],[0,0,0,0],[8.999999E+09,8.999999E+09,8.999999E+09,8.999999E+09,8.999999E+09,8.999999E+09]];
	LOCAL CONST Robtarget Tr_meulage_bavure_P8 :=[[-99.2814921875,-98.96675,23],[0.637806767491368,-0.68241616321174,0.260881077492864,-0.243827338368245],[0,0,0,0],[8.999999E+09,8.999999E+09,8.999999E+09,8.999999E+09,8.999999E+09,8.999999E+09]];
	LOCAL CONST Robtarget Tr_meulage_bavure_P9 :=[[-102.1833828125,-96.3584609375,23],[0.637504387013829,-0.680793507023223,0.263290641544285,-0.246548971622964],[0,0,0,0],[8.999999E+09,8.999999E+09,8.999999E+09,8.999999E+09,8.999999E+09,8.999999E+09]];
	LOCAL CONST Robtarget Tr_meulage_bavure_P10 :=[[-103.9701875,-94.720625,23],[0.63716665581841,-0.679088017653528,0.265812274943829,-0.249403190600624],[0,0,0,0],[8.999999E+09,8.999999E+09,8.999999E+09,8.999999E+09,8.999999E+09,8.999999E+09]];
	LOCAL CONST Robtarget Tr_meulage_bavure_P11 :=[[-107.26690625,-91.5796484375,23],[0.636810579408741,-0.677356695238329,0.2683498682862,-0.252286625804248],[0,0,0,0],[8.999999E+09,8.999999E+09,8.999999E+09,8.999999E+09,8.999999E+09,8.999999E+09]];
	LOCAL CONST Robtarget Tr_meulage_bavure_P12 :=[[-109.16,-89.716640625,23],[0.636483995915155,-0.675672630326605,0.270750256960323,-0.255046893584932],[0,0,0,0],[8.999999E+09,8.999999E+09,8.999999E+09,8.999999E+09,8.999999E+09,8.999999E+09]];
	LOCAL CONST Robtarget Tr_meulage_bavure_P13 :=[[-110.59384375,-88.204296875,23],[0.636234314913627,-0.674105609978111,0.272872480108507,-0.257542487216885],[0,0,0,0],[8.999999E+09,8.999999E+09,8.999999E+09,8.999999E+09,8.999999E+09,8.999999E+09]];
	LOCAL CONST Robtarget Tr_meulage_bavure_P14 :=[[-113.0693046875,-85.8259921875,23],[0.636078188142662,-0.672709572263584,0.274642880187524,-0.259687616794477],[0,0,0,0],[8.999999E+09,8.999999E+09,8.999999E+09,8.999999E+09,8.999999E+09,8.999999E+09]];
	LOCAL CONST Robtarget Tr_meulage_bavure_P15 :=[[-116.5336640625,-82.3804765625,23],[0.636028475705817,-0.671489248791908,0.27604879608022,-0.26147089518888],[0,0,0,0],[8.999999E+09,8.999999E+09,8.999999E+09,8.999999E+09,8.999999E+09,8.999999E+09]];
	LOCAL CONST Robtarget Tr_meulage_bavure_P16 :=[[-120.6395859375,-78.2647890625,23],[0.636042225763816,-0.670430237320022,0.27717565131788,-0.262958632200844],[0,0,0,0],[8.999999E+09,8.999999E+09,8.999999E+09,8.999999E+09,8.999999E+09,8.999999E+09]];
	LOCAL CONST Robtarget Tr_meulage_bavure_P17 :=[[-123.6929921875,-75.112546875,23],[0.636064252885398,-0.669468745135333,0.278175700838061,-0.264295563624356],[0,0,0,0],[8.999999E+09,8.999999E+09,8.999999E+09,8.999999E+09,8.999999E+09,8.999999E+09]];
	LOCAL CONST Robtarget Tr_meulage_bavure_P18 :=[[-125.3610546875,-73.3430625,23],[0.63601130581762,-0.668522856816576,0.279255586366879,-0.265674850651808],[0,0,0,0],[8.999999E+09,8.999999E+09,8.999999E+09,8.999999E+09,8.999999E+09,8.999999E+09]];
	LOCAL CONST Robtarget Tr_meulage_bavure_P19 :=[[-126.754453125,-71.9008203125,23],[0.635798331564058,-0.667510908550726,0.280619207298071,-0.267287352939766],[0,0,0,0],[8.999999E+09,8.999999E+09,8.999999E+09,8.999999E+09,8.999999E+09,8.999999E+09]];
	LOCAL CONST Robtarget Tr_meulage_bavure_P20 :=[[-127.72003125,-70.9483203125,23],[0.635386580587655,-0.666358440668368,0.282392524572639,-0.269267123549534],[0,0,0,0],[8.999999E+09,8.999999E+09,8.999999E+09,8.999999E+09,8.999999E+09,8.999999E+09]];
	LOCAL CONST Robtarget Tr_meulage_bavure_P21 :=[[-129.701046875,-68.8303203125,23],[0.63475462980096,-0.665061988110578,0.284598882750685,-0.27162950475549],[0,0,0,0],[8.999999E+09,8.999999E+09,8.999999E+09,8.999999E+09,8.999999E+09,8.999999E+09]];
	LOCAL CONST Robtarget Tr_meulage_bavure_P22 :=[[-133.266140625,-64.94608984375,23],[0.633945287803024,-0.663644335818577,0.287144685936053,-0.274294544143602],[0,0,0,0],[8.999999E+09,8.999999E+09,8.999999E+09,8.999999E+09,8.999999E+09,8.999999E+09]];
	LOCAL CONST Robtarget Tr_meulage_bavure_P23 :=[[-136.61690625,-61.2477890625,23],[0.633026518144594,-0.662149956801891,0.289882991067473,-0.277133024958704],[0,0,0,0],[8.999999E+09,8.999999E+09,8.999999E+09,8.999999E+09,8.999999E+09,8.999999E+09]];
	LOCAL CONST Robtarget Tr_meulage_bavure_P24 :=[[-139.611046875,-57.939515625,23],[0.632037253703891,-0.660627160403708,0.29270800877669,-0.280040508615025],[0,0,0,0],[8.999999E+09,8.999999E+09,8.999999E+09,8.999999E+09,8.999999E+09,8.999999E+09]];
	LOCAL CONST Robtarget Tr_meulage_bavure_P25 :=[[-141.01071875,-56.387984375,23],[0.630993537474336,-0.65907023159802,0.295600962951187,-0.283008226363277],[0,0,0,0],[8.999999E+09,8.999999E+09,8.999999E+09,8.999999E+09,8.999999E+09,8.999999E+09]];
	LOCAL CONST Robtarget Tr_meulage_bavure_P26 :=[[-142.894984375,-54.19334375,23],[0.629870537950577,-0.657440992412034,0.298627866258112,-0.286104603968998],[0,0,0,0],[8.999999E+09,8.999999E+09,8.999999E+09,8.999999E+09,8.999999E+09,8.999999E+09]];
	LOCAL CONST Robtarget Tr_meulage_bavure_P27 :=[[-148.83384375,-47.14578125,23],[0.628625836707171,-0.655700367057112,0.301874794905319,-0.28941007975924],[0,0,0,0],[8.999999E+09,8.999999E+09,8.999999E+09,8.999999E+09,8.999999E+09,8.999999E+09]];
	LOCAL CONST Robtarget Tr_meulage_bavure_P28 :=[[-149.9493125,-45.86146484375,23],[0.627264437632511,-0.653822066989345,0.305349554865432,-0.292946546903753],[0,0,0,0],[8.999999E+09,8.999999E+09,8.999999E+09,8.999999E+09,8.999999E+09,8.999999E+09]];
	LOCAL CONST Robtarget Tr_meulage_bavure_P29 :=[[-150.858,-44.7060234375,23],[0.625818835765137,-0.651864912808947,0.308948303181207,-0.296603887721664],[0,0,0,0],[8.999999E+09,8.999999E+09,8.999999E+09,8.999999E+09,8.999999E+09,8.999999E+09]];
	LOCAL CONST Robtarget Tr_meulage_bavure_P30 :=[[-152.825828125,-42.34896875,23],[0.624396411650755,-0.649932169813015,0.312439961374253,-0.30016423220674],[0,0,0,0],[8.999999E+09,8.999999E+09,8.999999E+09,8.999999E+09,8.999999E+09,8.999999E+09]];
	LOCAL CONST Robtarget Tr_meulage_bavure_P31 :=[[-153.0646875,-42.045625,23],[0.623128571603386,-0.648151082205295,0.315555833054265,-0.303373489469759],[0,0,0,0],[8.999999E+09,8.999999E+09,8.999999E+09,8.999999E+09,8.999999E+09,8.999999E+09]];
	LOCAL CONST Robtarget Tr_meulage_bavure_P32 :=[[-153.298609375,-41.76766796875,23],[0.622101615019679,-0.646639672197605,0.318104347838139,-0.306033231555911],[0,0,0,0],[8.999999E+09,8.999999E+09,8.999999E+09,8.999999E+09,8.999999E+09,8.999999E+09]];
	LOCAL CONST Robtarget Tr_meulage_bavure_P33 :=[[-155.45503125,-39.067046875,23],[0.621360991750904,-0.64542809871959,0.320022227139241,-0.308089047923467],[0,0,0,0],[8.999999E+09,8.999999E+09,8.999999E+09,8.999999E+09,8.999999E+09,8.999999E+09]];
	LOCAL CONST Robtarget Tr_meulage_bavure_P34 :=[[-155.83853125,-38.5523359375,23],[0.620857143190513,-0.644497282892196,0.321402172718058,-0.30961315131306],[0,0,0,0],[8.999999E+09,8.999999E+09,8.999999E+09,8.999999E+09,8.999999E+09,8.999999E+09]];
	LOCAL CONST Robtarget Tr_meulage_bavure_P35 :=[[-159.17671875,-34.22415234375,23],[0.620510879787186,-0.643752048014424,0.322428700014739,-0.310788162821195],[0,0,0,0],[8.999999E+09,8.999999E+09,8.999999E+09,8.999999E+09,8.999999E+09,8.999999E+09]];
	LOCAL CONST Robtarget Tr_meulage_bavure_P36 :=[[-159.614484375,-33.6722421875,23],[0.620218750642947,-0.643101969403024,0.323307071459069,-0.311802976004742],[0,0,0,0],[8.999999E+09,8.999999E+09,8.999999E+09,8.999999E+09,8.999999E+09,8.999999E+09]];
	LOCAL CONST Robtarget Tr_meulage_bavure_P37 :=[[-164.3065,-27.351958984375,23],[0.619890611494999,-0.642478796336214,0.324204798642968,-0.312806449063313],[0,0,0,0],[8.999999E+09,8.999999E+09,8.999999E+09,8.999999E+09,8.999999E+09,8.999999E+09]];
	LOCAL CONST Robtarget Tr_meulage_bavure_P38 :=[[-164.679265625,-26.8167109375,23],[0.619490877937617,-0.641827151607868,0.325209214013912,-0.313891584359098],[0,0,0,0],[8.999999E+09,8.999999E+09,8.999999E+09,8.999999E+09,8.999999E+09,8.999999E+09]];
	LOCAL CONST Robtarget Tr_meulage_bavure_P39 :=[[-165.112953125,-26.228423828125,23],[0.618991396534955,-0.641149503195034,0.326352128978416,-0.315073409667847],[0,0,0,0],[8.999999E+09,8.999999E+09,8.999999E+09,8.999999E+09,8.999999E+09,8.999999E+09]];
	LOCAL CONST Robtarget Tr_meulage_bavure_P40 :=[[-168.454140625,-21.6435234375,23],[0.618397504728911,-0.64046456000676,0.327611247886881,-0.316323479650824],[0,0,0,0],[8.999999E+09,8.999999E+09,8.999999E+09,8.999999E+09,8.999999E+09,8.999999E+09]];
	LOCAL CONST Robtarget Tr_meulage_bavure_P41 :=[[-170.152671875,-19.283935546875,23],[0.617747448699429,-0.639791211933322,0.328924175351972,-0.317591217805631],[0,0,0,0],[8.999999E+09,8.999999E+09,8.999999E+09,8.999999E+09,8.999999E+09,8.999999E+09]];
	LOCAL CONST Robtarget Tr_meulage_bavure_P42 :=[[-170.8105625,-18.345611328125,23],[0.617049734714428,-0.639180094712443,0.330242079273067,-0.318808093513398],[0,0,0,0],[8.999999E+09,8.999999E+09,8.999999E+09,8.999999E+09,8.999999E+09,8.999999E+09]];
	LOCAL CONST Robtarget Tr_meulage_bavure_P43 :=[[-172.78721875,-15.3552548828125,23],[0.616334210054334,-0.63864321688449,0.331520205610946,-0.319939582289854],[0,0,0,0],[8.999999E+09,8.999999E+09,8.999999E+09,8.999999E+09,8.999999E+09,8.999999E+09]];
	LOCAL CONST Robtarget Tr_meulage_bavure_P44 :=[[-175.414875,-11.6484072265625,23],[0.615589801404961,-0.638176417656608,0.33277624531692,-0.320998484273606],[0,0,0,0],[8.999999E+09,8.999999E+09,8.999999E+09,8.999999E+09,8.999999E+09,8.999999E+09]];
	LOCAL CONST Robtarget Tr_meulage_bavure_P45 :=[[-178.3580625,-7.5121767578125,23],[0.614779802406032,-0.637751433947501,0.33407650057798,-0.322043156755546],[0,0,0,0],[8.999999E+09,8.999999E+09,8.999999E+09,8.999999E+09,8.999999E+09,8.999999E+09]];
	LOCAL CONST Robtarget Tr_meulage_bavure_P46 :=[[-178.55940625,-7.215087890625,23],[0.613864826875311,-0.637308017287822,0.335512871936265,-0.323171128337741],[0,0,0,0],[8.999999E+09,8.999999E+09,8.999999E+09,8.999999E+09,8.999999E+09,8.999999E+09]];
	LOCAL CONST Robtarget Tr_meulage_bavure_P47 :=[[-178.75059375,-6.9400634765625,23],[0.612782220386535,-0.636811484649985,0.337184944276332,-0.324461703055069],[0,0,0,0],[8.999999E+09,8.999999E+09,8.999999E+09,8.999999E+09,8.999999E+09,8.999999E+09]];
	LOCAL CONST Robtarget Tr_meulage_bavure_P48 :=[[-180.717390625,-3.98046875,23],[0.611519180077081,-0.63621354458658,0.339140039042336,-0.325976459273975],[0,0,0,0],[8.999999E+09,8.999999E+09,8.999999E+09,8.999999E+09,8.999999E+09,8.999999E+09]];
	LOCAL CONST Robtarget Tr_meulage_bavure_P49 :=[[-183.206828125,-0.16949462890625,23],[0.610065448834155,-0.635516855483889,0.341384150982413,-0.327712276231251],[0,0,0,0],[8.999999E+09,8.999999E+09,8.999999E+09,8.999999E+09,8.999999E+09,8.999999E+09]];
	LOCAL CONST Robtarget Tr_meulage_bavure_P50 :=[[-184.33109375,1.59613037109375,23],[0.608453010454663,-0.634744382144604,0.343857968834926,-0.329615231251898],[0,0,0,0],[8.999999E+09,8.999999E+09,8.999999E+09,8.999999E+09,8.999999E+09,8.999999E+09]];
	LOCAL CONST Robtarget Tr_meulage_bavure_P51 :=[[-185.79925,3.86856079101563,23],[0.606741149397428,-0.633947543958269,0.346451199835319,-0.331582953828805],[0,0,0,0],[8.999999E+09,8.999999E+09,8.999999E+09,8.999999E+09,8.999999E+09,8.999999E+09]];
	LOCAL CONST Robtarget Tr_meulage_bavure_P52 :=[[-186.629203125,5.2182919921875,23],[0.604999265121601,-0.633204720335686,0.349026211815068,-0.333479196971792],[0,0,0,0],[8.999999E+09,8.999999E+09,8.999999E+09,8.999999E+09,8.999999E+09,8.999999E+09]];
	LOCAL CONST Robtarget Tr_meulage_bavure_P53 :=[[-188.1745625,7.6268310546875,23],[0.603304686627718,-0.63259519792822,0.351439547794507,-0.335167144716155],[0,0,0,0],[8.999999E+09,8.999999E+09,8.999999E+09,8.999999E+09,8.999999E+09,8.999999E+09]];
	LOCAL CONST Robtarget Tr_meulage_bavure_P54 :=[[-189.39925,9.66665625,23],[0.601718435413318,-0.632183459076313,0.353580289179188,-0.336541197564308],[0,0,0,0],[8.999999E+09,8.999999E+09,8.999999E+09,8.999999E+09,8.999999E+09,8.999999E+09]];
	LOCAL CONST Robtarget Tr_meulage_bavure_P55 :=[[-190.449453125,11.194671875,23],[0.600260751247743,-0.631981502414589,0.355421769858607,-0.337582251648201],[0,0,0,0],[8.999999E+09,8.999999E+09,8.999999E+09,8.999999E+09,8.999999E+09,8.999999E+09]];
	LOCAL CONST Robtarget Tr_meulage_bavure_P56 :=[[-193.0021875,15.32894921875,23],[0.598899171682936,-0.63195151945624,0.357031066493161,-0.33835761669157],[0,0,0,0],[8.999999E+09,8.999999E+09,8.999999E+09,8.999999E+09,8.999999E+09,8.999999E+09]];
	LOCAL CONST Robtarget Tr_meulage_bavure_P57 :=[[-193.809484375,16.6774296875,23],[0.597540305255729,-0.632016536080522,0.35857025621071,-0.339010402608319],[0,0,0,0],[8.999999E+09,8.999999E+09,8.999999E+09,8.999999E+09,8.999999E+09,8.999999E+09]];
	LOCAL CONST Robtarget Tr_meulage_bavure_P58 :=[[-194.320375,17.45446875,23],[0.596087253125083,-0.632056195294275,0.360232029291838,-0.339732008683613],[0,0,0,0],[8.999999E+09,8.999999E+09,8.999999E+09,8.999999E+09,8.999999E+09,8.999999E+09]];
	LOCAL CONST Robtarget Tr_meulage_bavure_P59 :=[[-197.90896875,23.49331640625,23],[0.594443672767175,-0.631967083053523,0.362194851849808,-0.340689323486059],[0,0,0,0],[8.999999E+09,8.999999E+09,8.999999E+09,8.999999E+09,8.999999E+09,8.999999E+09]];
	LOCAL CONST Robtarget Tr_meulage_bavure_P60 :=[[-199.941640625,26.863494140625,23],[0.592567900826204,-0.631688664795584,0.364542926625118,-0.341966618731699],[0,0,0,0],[8.999999E+09,8.999999E+09,8.999999E+09,8.999999E+09,8.999999E+09,8.999999E+09]];
	LOCAL CONST Robtarget Tr_meulage_bavure_P61 :=[[-202.821984375,31.87448046875,23],[0.590486245475775,-0.631235550397876,0.367231006360412,-0.343524470431632],[0,0,0,0],[8.999999E+09,8.999999E+09,8.999999E+09,8.999999E+09,8.999999E+09,8.999999E+09]];
	LOCAL CONST Robtarget Tr_meulage_bavure_P62 :=[[-203.23153125,32.622771484375,23],[0.588271780316929,-0.630692396132256,0.370115589713001,-0.345221471225506],[0,0,0,0],[8.999999E+09,8.999999E+09,8.999999E+09,8.999999E+09,8.999999E+09,8.999999E+09]];
	LOCAL CONST Robtarget Tr_meulage_bavure_P63 :=[[-203.5151875,33.11737109375,23],[0.586062930618858,-0.630157402966473,0.372973707596959,-0.346875341127563],[0,0,0,0],[8.999999E+09,8.999999E+09,8.999999E+09,8.999999E+09,8.999999E+09,8.999999E+09]];
	LOCAL CONST Robtarget Tr_meulage_bavure_P64 :=[[-203.923171875,33.89599609375,23],[0.583965838177081,-0.629734488890245,0.375620731196099,-0.348320886023202],[0,0,0,0],[8.999999E+09,8.999999E+09,8.999999E+09,8.999999E+09,8.999999E+09,8.999999E+09]];
	LOCAL CONST Robtarget Tr_meulage_bavure_P65 :=[[-208.35253125,42.4410078125,23],[0.58203306738214,-0.629463127274778,0.377976512360161,-0.349495974196045],[0,0,0,0],[8.999999E+09,8.999999E+09,8.999999E+09,8.999999E+09,8.999999E+09,8.999999E+09]];
	LOCAL CONST Robtarget Tr_meulage_bavure_P66 :=[[-208.638125,42.962890625,23],[0.580265584280528,-0.62930320731391,0.380068885149213,-0.350452518189609],[0,0,0,0],[8.999999E+09,8.999999E+09,8.999999E+09,8.999999E+09,8.999999E+09,8.999999E+09]];
	LOCAL CONST Robtarget Tr_meulage_bavure_P67 :=[[-209.91159375,45.507203125,23],[0.578614619733604,-0.629185240662071,0.381998289005791,-0.351295263219129],[0,0,0,0],[8.999999E+09,8.999999E+09,8.999999E+09,8.999999E+09,8.999999E+09,8.999999E+09]];
	LOCAL CONST Robtarget Tr_meulage_bavure_P68 :=[[-211.25371875,48.042296875,23],[0.577043422214005,-0.629023966515235,0.383859535935959,-0.352138602115729],[0,0,0,0],[8.999999E+09,8.999999E+09,8.999999E+09,8.999999E+09,8.999999E+09,8.999999E+09]];
	LOCAL CONST Robtarget Tr_meulage_bavure_P69 :=[[-211.85778125,49.3566875,23],[0.575527810220992,-0.628791216350221,0.385697104521361,-0.353025621544496],[0,0,0,0],[8.999999E+09,8.999999E+09,8.999999E+09,8.999999E+09,8.999999E+09,8.999999E+09]];
	LOCAL CONST Robtarget Tr_meulage_bavure_P70 :=[[-212.5911875,50.68365625,23],[0.574090637312713,-0.628470953855987,0.387495004701937,-0.353965848127013],[0,0,0,0],[8.999999E+09,8.999999E+09,8.999999E+09,8.999999E+09,8.999999E+09,8.999999E+09]];
	LOCAL CONST Robtarget Tr_meulage_bavure_P71 :=[[-214.616,54.92309375,23],[0.572737548397397,-0.628046056014274,0.389256964314139,-0.354977278024377],[0,0,0,0],[8.999999E+09,8.999999E+09,8.999999E+09,8.999999E+09,8.999999E+09,8.999999E+09]];
	LOCAL CONST Robtarget Tr_meulage_bavure_P72 :=[[-215.722828125,57.05776953125,23],[0.571433488449121,-0.627468270771563,0.391050021751212,-0.356128092043003],[0,0,0,0],[8.999999E+09,8.999999E+09,8.999999E+09,8.999999E+09,8.999999E+09,8.999999E+09]];
	LOCAL CONST Robtarget Tr_meulage_bavure_P73 :=[[-216.546703125,58.9495234375,23],[0.570105343438099,-0.626639386758814,0.393011125237221,-0.357554515823304],[0,0,0,0],[8.999999E+09,8.999999E+09,8.999999E+09,8.999999E+09,8.999999E+09,8.999999E+09]];
	LOCAL CONST Robtarget Tr_meulage_bavure_P74 :=[[-217.575921875,60.988984375,23],[0.568667118475947,-0.625466341776934,0.395284336157361,-0.359388170725023],[0,0,0,0],[8.999999E+09,8.999999E+09,8.999999E+09,8.999999E+09,8.999999E+09,8.999999E+09]];
	LOCAL CONST Robtarget Tr_meulage_bavure_P75 :=[[-218.500390625,63.14721875,23],[0.567075129138539,-0.623901788681195,0.397935296920799,-0.361690275591522],[0,0,0,0],[8.999999E+09,8.999999E+09,8.999999E+09,8.999999E+09,8.999999E+09,8.999999E+09]];
	LOCAL CONST Robtarget Tr_meulage_bavure_P76 :=[[-220.6359375,68.1213984375,23],[0.565352211910123,-0.62196126765576,0.400916845328114,-0.364426592274115],[0,0,0,0],[8.999999E+09,8.999999E+09,8.999999E+09,8.999999E+09,8.999999E+09,8.999999E+09]];
	LOCAL CONST Robtarget Tr_meulage_bavure_P77 :=[[-221.501671875,70.223359375,23],[0.563576734027623,-0.619736487761388,0.404078927588143,-0.367461795128627],[0,0,0,0],[8.999999E+09,8.999999E+09,8.999999E+09,8.999999E+09,8.999999E+09,8.999999E+09]];
	LOCAL CONST Robtarget Tr_meulage_bavure_P78 :=[[-221.745359375,70.870328125,23],[0.561836089087529,-0.617339369283921,0.407256206351076,-0.37064092396751],[0,0,0,0],[8.999999E+09,8.999999E+09,8.999999E+09,8.999999E+09,8.999999E+09,8.999999E+09]];
	LOCAL CONST Robtarget Tr_meulage_bavure_P79 :=[[-222.486640625,72.465328125,23],[0.560126777965476,-0.61478423122543,0.410439269039751,-0.373949124979169],[0,0,0,0],[8.999999E+09,8.999999E+09,8.999999E+09,8.999999E+09,8.999999E+09,8.999999E+09]];
	LOCAL CONST Robtarget Tr_meulage_bavure_P80 :=[[-222.990421875,73.6807890625,23],[0.558309536302779,-0.61192149105019,0.413846919633065,-0.377588767807665],[0,0,0,0],[8.999999E+09,8.999999E+09,8.999999E+09,8.999999E+09,8.999999E+09,8.999999E+09]];
	LOCAL CONST Robtarget Tr_meulage_bavure_P81 :=[[-224.275796875,76.966890625,23],[0.556005864862951,-0.608323970498805,0.418073555705783,-0.382117687596497],[0,0,0,0],[8.999999E+09,8.999999E+09,8.999999E+09,8.999999E+09,8.999999E+09,8.999999E+09]];
	LOCAL CONST Robtarget Tr_meulage_bavure_P82 :=[[-225.08675,78.7561640625,23],[0.552536485772631,-0.603291624405466,0.42410737042647,-0.388427066721913],[0,0,0,0],[8.999999E+09,8.999999E+09,8.999999E+09,8.999999E+09,8.999999E+09,8.999999E+09]];
	LOCAL CONST Robtarget Tr_meulage_bavure_P83 :=[[-225.64590625,79.798890625,23],[0.547042449373018,-0.595881458186565,0.433103958325402,-0.397606347605631],[0,0,0,0],[8.999999E+09,8.999999E+09,8.999999E+09,8.999999E+09,8.999999E+09,8.999999E+09]];
	LOCAL CONST Robtarget Tr_meulage_bavure_P84 :=[[-225.846171875,80.3101484375,23],[0.538528629534617,-0.585048450894237,0.446151069155635,-0.410675600406337],[0,0,0,0],[8.999999E+09,8.999999E+09,8.999999E+09,8.999999E+09,8.999999E+09,8.999999E+09]];
	LOCAL CONST Robtarget Tr_meulage_bavure_P85 :=[[-227.168125,83.241515625,23],[0.526109946657191,-0.569869496956498,0.46380227653179,-0.428187492520327],[0,0,0,0],[8.999999E+09,8.999999E+09,8.999999E+09,8.999999E+09,8.999999E+09,8.999999E+09]];
	LOCAL CONST Robtarget Tr_meulage_bavure_P86 :=[[-227.25865625,83.4700625,23],[0.509064114791511,-0.549613059145104,0.485974174609354,-0.45012033264612],[0,0,0,0],[8.999999E+09,8.999999E+09,8.999999E+09,8.999999E+09,8.999999E+09,8.999999E+09]];
	LOCAL CONST Robtarget Tr_meulage_bavure_P87 :=[[-227.48228125,84.181734375,23],[0.486761621251007,-0.523655575018831,0.512103316451494,-0.476023272653943],[0,0,0,0],[8.999999E+09,8.999999E+09,8.999999E+09,8.999999E+09,8.999999E+09,8.999999E+09]];
	LOCAL CONST Robtarget Tr_meulage_bavure_P88 :=[[-228.1584375,86.6586875,23],[0.458405590863769,-0.49122954187092,0.541495238875229,-0.505312534708555],[0,0,0,0],[8.999999E+09,8.999999E+09,8.999999E+09,8.999999E+09,8.999999E+09,8.999999E+09]];
	LOCAL CONST Robtarget Tr_meulage_bavure_P89 :=[[-227.72525,89.4899609375,23],[0.422874111002271,-0.451252407976164,0.573412444553177,-0.537351764648914],[0,0,0,0],[8.999999E+09,8.999999E+09,8.999999E+09,8.999999E+09,8.999999E+09,8.999999E+09]];
	LOCAL CONST Robtarget Tr_meulage_bavure_P90 :=[[-227.624265625,89.8831484375,23],[0.379415432646327,-0.403050310237239,0.6064062600967,-0.570846585873122],[0,0,0,0],[8.999999E+09,8.999999E+09,8.999999E+09,8.999999E+09,8.999999E+09,8.999999E+09]];
	LOCAL CONST Robtarget Tr_meulage_bavure_P91 :=[[-226.95615625,90.7658046875,23],[0.329269230078473,-0.348094514473986,0.637652527792685,-0.603167668991176],[0,0,0,0],[8.999999E+09,8.999999E+09,8.999999E+09,8.999999E+09,8.999999E+09,8.999999E+09]];
	LOCAL CONST Robtarget Tr_meulage_bavure_P92 :=[[-226.279703125,91.630984375,23],[0.277049947022601,-0.291383831761022,0.663547958543036,-0.630906408397004],[0,0,0,0],[8.999999E+09,8.999999E+09,8.999999E+09,8.999999E+09,8.999999E+09,8.999999E+09]];
	LOCAL CONST Robtarget Tr_meulage_bavure_P93 :=[[-223.598421875,93.2830234375,23],[0.229382700432276,-0.239933594820948,0.681837171449315,-0.651853908823666],[0,0,0,0],[8.999999E+09,8.999999E+09,8.999999E+09,8.999999E+09,8.999999E+09,8.999999E+09]];
	LOCAL CONST Robtarget Tr_meulage_bavure_P94 :=[[-223.413234375,93.4259609375,23],[0.191279382349789,-0.198929466566882,0.69283810276071,-0.666194137307016],[0,0,0,0],[8.999999E+09,8.999999E+09,8.999999E+09,8.999999E+09,8.999999E+09,8.999999E+09]];
	LOCAL CONST Robtarget Tr_meulage_bavure_P95 :=[[-222.693234375,93.70434375,23],[0.164241603691448,-0.169780969018371,0.698393634161807,-0.675607467349428],[0,0,0,0],[8.999999E+09,8.999999E+09,8.999999E+09,8.999999E+09,8.999999E+09,8.999999E+09]];
	LOCAL CONST Robtarget Tr_meulage_bavure_P96 :=[[-219.287515625,94.9596875,23],[0.14707344188631,-0.151074231244549,0.700423428233405,-0.681874622293092],[0,0,0,0],[8.999999E+09,8.999999E+09,8.999999E+09,8.999999E+09,8.999999E+09,8.999999E+09]];
	LOCAL CONST Robtarget Tr_meulage_bavure_P97 :=[[-215.06440625,96.426359375,23],[0.137381711164586,-0.140194089509967,0.700340279019509,-0.686291028854988],[0,0,0,0],[8.999999E+09,8.999999E+09,8.999999E+09,8.999999E+09,8.999999E+09,8.999999E+09]];
	LOCAL CONST Robtarget Tr_meulage_bavure_P98 :=[[-207.5475,99.17565625,23],[0.13273983119406,-0.134537975724687,0.699018492163638,-0.689675878884966],[0,0,0,0],[8.999999E+09,8.999999E+09,8.999999E+09,8.999999E+09,8.999999E+09,8.999999E+09]];
	LOCAL CONST Robtarget Tr_meulage_bavure_P99 :=[[-202.719625,100.9839765625,23],[0.131120472537897,-0.131965197860097,0.696990667727135,-0.692529145477984],[0,0,0,0],[8.999999E+09,8.999999E+09,8.999999E+09,8.999999E+09,8.999999E+09,8.999999E+09]];
	LOCAL CONST Robtarget Tr_meulage_bavure_P100 :=[[-200.20753125,101.9860859375,23],[0.131080127359178,-0.130972963633238,0.694576953171572,-0.695145264769547],[0,0,0,0],[8.999999E+09,8.999999E+09,8.999999E+09,8.999999E+09,8.999999E+09,8.999999E+09]];
	LOCAL CONST Robtarget Tr_meulage_bavure_P101 :=[[-192.306046875,105.0720859375,23],[0.131682131327459,-0.130606241417043,0.691982762439855,-0.697683081691163],[0,0,0,0],[8.999999E+09,8.999999E+09,8.999999E+09,8.999999E+09,8.999999E+09,8.999999E+09]];
	LOCAL CONST Robtarget Tr_meulage_bavure_P102 :=[[-188.0050625,106.8087734375,23],[0.13233403678279,-0.13027196535847,0.689331095995641,-0.700242499312817],[0,0,0,0],[8.999999E+09,8.999999E+09,8.999999E+09,8.999999E+09,8.999999E+09,8.999999E+09]];
	LOCAL CONST Robtarget Tr_meulage_bavure_P103 :=[[-184.288375,108.2283046875,23],[0.132823438924978,-0.129760966041877,0.686659205570545,-0.702864966525754],[0,0,0,0],[8.999999E+09,8.999999E+09,8.999999E+09,8.999999E+09,8.999999E+09,8.999999E+09]];
	LOCAL CONST Robtarget Tr_meulage_bavure_P104 :=[[-182.750859375,108.85690625,23],[0.13313338519322,-0.129069815066325,0.683993358343489,-0.705527866443086],[0,0,0,0],[8.999999E+09,8.999999E+09,8.999999E+09,8.999999E+09,8.999999E+09,8.999999E+09]];
	LOCAL CONST Robtarget Tr_meulage_bavure_P105 :=[[-175.827140625,111.3243125,23],[0.133373245574566,-0.128317012483931,0.681337297423167,-0.708184869092951],[0,0,0,0],[8.999999E+09,8.999999E+09,8.999999E+09,8.999999E+09,8.999999E+09,8.999999E+09]];
	LOCAL CONST Robtarget Tr_meulage_bavure_P106 :=[[-173.832390625,112.04565625,23],[0.133682255185474,-0.127640356807583,0.678675057926722,-0.710800365581447],[0,0,0,0],[8.999999E+09,8.999999E+09,8.999999E+09,8.999999E+09,8.999999E+09,8.999999E+09]];
	LOCAL CONST Robtarget Tr_meulage_bavure_P107 :=[[-173.1296875,112.2573515625,23],[0.134076912789235,-0.127062944677629,0.676029083628304,-0.713346386852441],[0,0,0,0],[8.999999E+09,8.999999E+09,8.999999E+09,8.999999E+09,8.999999E+09,8.999999E+09]];
	LOCAL CONST Robtarget Tr_meulage_bavure_P108 :=[[-172.613578125,112.4072578125,23],[0.134432333869445,-0.126476365347038,0.673452857807962,-0.715816264783991],[0,0,0,0],[8.999999E+09,8.999999E+09,8.999999E+09,8.999999E+09,8.999999E+09,8.999999E+09]];
	LOCAL CONST Robtarget Tr_meulage_bavure_P109 :=[[-171.29321875,112.818390625,23],[0.134539619007079,-0.125695135861112,0.671009231403881,-0.718224501885768],[0,0,0,0],[8.999999E+09,8.999999E+09,8.999999E+09,8.999999E+09,8.999999E+09,8.999999E+09]];
	LOCAL CONST Robtarget Tr_meulage_bavure_P110 :=[[-166.94565625,114.5949375,23],[0.134241897356325,-0.124585901160045,0.668747756055616,-0.72057886799218],[0,0,0,0],[8.999999E+09,8.999999E+09,8.999999E+09,8.999999E+09,8.999999E+09,8.999999E+09]];
	LOCAL CONST Robtarget Tr_meulage_bavure_P111 :=[[-166.10790625,114.9887421875,23],[0.133581411360778,-0.123206818280231,0.666696753272334,-0.722835752881838],[0,0,0,0],[8.999999E+09,8.999999E+09,8.999999E+09,8.999999E+09,8.999999E+09,8.999999E+09]];
	LOCAL CONST Robtarget Tr_meulage_bavure_P112 :=[[-165.576859375,115.1702890625,23],[0.132827466732656,-0.121818114896886,0.66483606219904,-0.724920837998211],[0,0,0,0],[8.999999E+09,8.999999E+09,8.999999E+09,8.999999E+09,8.999999E+09,8.999999E+09]];
	LOCAL CONST Robtarget Tr_meulage_bavure_P113 :=[[-156.145875,118.6306171875,23],[0.132418808650214,-0.120830439053086,0.663126582992309,-0.726724431296238],[0,0,0,0],[8.999999E+09,8.999999E+09,8.999999E+09,8.999999E+09,8.999999E+09,8.999999E+09]];
	LOCAL CONST Robtarget Tr_meulage_bavure_P114 :=[[-154.747203125,119.1098359375,23],[0.1328017382441,-0.120647306075702,0.661512014906197,-0.72815505216318],[0,0,0,0],[8.999999E+09,8.999999E+09,8.999999E+09,8.999999E+09,8.999999E+09,8.999999E+09]];
	LOCAL CONST Robtarget Tr_meulage_bavure_P115 :=[[-152.75003125,119.97128125,23],[0.134256375549463,-0.121520896169291,0.659973121674901,-0.729138790687494],[0,0,0,0],[8.999999E+09,8.999999E+09,8.999999E+09,8.999999E+09,8.999999E+09,8.999999E+09]];
	LOCAL CONST Robtarget Tr_meulage_bavure_P116 :=[[-150.449125,120.91678125,23],[0.136792337727519,-0.123453710778388,0.658513145612816,-0.729662575913826],[0,0,0,0],[8.999999E+09,8.999999E+09,8.999999E+09,8.999999E+09,8.999999E+09,8.999999E+09]];
	LOCAL CONST Robtarget Tr_meulage_bavure_P117 :=[[-147.3660625,122.18359375,23],[0.140112147120974,-0.126176495399087,0.657183038161223,-0.729766080734875],[0,0,0,0],[8.999999E+09,8.999999E+09,8.999999E+09,8.999999E+09,8.999999E+09,8.999999E+09]];
	LOCAL CONST Robtarget Tr_meulage_bavure_P118 :=[[-143.346625,123.634,23],[0.143707577841555,-0.129232929615318,0.65606046533876,-0.729542080892833],[0,0,0,0],[8.999999E+09,8.999999E+09,8.999999E+09,8.999999E+09,8.999999E+09,8.999999E+09]];
	LOCAL CONST Robtarget Tr_meulage_bavure_P119 :=[[-139.0588125,125.2717578125,23],[0.146992982254647,-0.132100251013836,0.655240337558996,-0.729110887921405],[0,0,0,0],[8.999999E+09,8.999999E+09,8.999999E+09,8.999999E+09,8.999999E+09,8.999999E+09]];
	LOCAL CONST Robtarget Tr_meulage_bavure_P120 :=[[-138.84503125,125.374359375,23],[0.149511412257956,-0.134361714303622,0.654775265393915,-0.728603197331958],[0,0,0,0],[8.999999E+09,8.999999E+09,8.999999E+09,8.999999E+09,8.999999E+09,8.999999E+09]];
	LOCAL CONST Robtarget Tr_meulage_bavure_P121 :=[[-138.535,125.5080234375,23],[0.15107800638927,-0.135846789215805,0.654683484861015,-0.728086959432345],[0,0,0,0],[8.999999E+09,8.999999E+09,8.999999E+09,8.999999E+09,8.999999E+09,8.999999E+09]];
	LOCAL CONST Robtarget Tr_meulage_bavure_P122 :=[[-130.47903125,128.7274765625,23],[0.151809998160049,-0.136647480869511,0.654910808337613,-0.727580252311205],[0,0,0,0],[8.999999E+09,8.999999E+09,8.999999E+09,8.999999E+09,8.999999E+09,8.999999E+09]];
	LOCAL CONST Robtarget Tr_meulage_bavure_P123 :=[[-129.8134453125,129.150546875,23],[0.152058952391352,-0.137062838614828,0.655351152794026,-0.727053450442284],[0,0,0,0],[8.999999E+09,8.999999E+09,8.999999E+09,8.999999E+09,8.999999E+09,8.999999E+09]];
	LOCAL CONST Robtarget Tr_meulage_bavure_P124 :=[[-129.0030234375,129.4828828125,23],[0.152208361672442,-0.137417972611912,0.655882602509751,-0.726475689314693],[0,0,0,0],[8.999999E+09,8.999999E+09,8.999999E+09,8.999999E+09,8.999999E+09,8.999999E+09]];
	LOCAL CONST Robtarget Tr_meulage_bavure_P125 :=[[-126.592984375,130.564484375,23],[0.15251509699267,-0.137921016409783,0.656395840750138,-0.725852215445905],[0,0,0,0],[8.999999E+09,8.999999E+09,8.999999E+09,8.999999E+09,8.999999E+09,8.999999E+09]];
	LOCAL CONST Robtarget Tr_meulage_bavure_P126 :=[[-124.177125,131.57909375,23],[0.153046713690908,-0.138614134022577,0.656827891457415,-0.72521717180524],[0,0,0,0],[8.999999E+09,8.999999E+09,8.999999E+09,8.999999E+09,8.999999E+09,8.999999E+09]];
	LOCAL CONST Robtarget Tr_meulage_bavure_P127 :=[[-119.71090625,133.578453125,23],[0.153702983180222,-0.139388342403775,0.657150597900017,-0.724637409083383],[0,0,0,0],[8.999999E+09,8.999999E+09,8.999999E+09,8.999999E+09,8.999999E+09,8.999999E+09]];
	LOCAL CONST Robtarget Tr_meulage_bavure_P128 :=[[-115.9326171875,134.801296875,23],[0.154317845254057,-0.140073505006325,0.657348232467839,-0.724195220298226],[0,0,0,0],[8.999999E+09,8.999999E+09,8.999999E+09,8.999999E+09,8.999999E+09,8.999999E+09]];
	LOCAL CONST Robtarget Tr_meulage_bavure_P129 :=[[-112.962375,136.22165625,23],[0.154644517681236,-0.140428386725702,0.657429137445656,-0.723983335851189],[0,0,0,0],[8.999999E+09,8.999999E+09,8.999999E+09,8.999999E+09,8.999999E+09,8.999999E+09]];
	LOCAL CONST Robtarget Tr_meulage_bavure_P130 :=[[-108.40240625,137.73059375,23],[0.154400421223228,-0.14018531385552,0.657423463024845,-0.724087686658004],[0,0,0,0],[8.999999E+09,8.999999E+09,8.999999E+09,8.999999E+09,8.999999E+09,8.999999E+09]];
	LOCAL CONST Robtarget Tr_meulage_bavure_P131 :=[[-108.1422109375,137.8111875,23],[0.153207405873798,-0.13899816301184,0.657393846467356,-0.724596668562318],[0,0,0,0],[8.999999E+09,8.999999E+09,8.999999E+09,8.999999E+09,8.999999E+09,8.999999E+09]];
	LOCAL CONST Robtarget Tr_meulage_bavure_P132 :=[[-107.3793359375,138.154171875,23],[0.150693131219862,-0.136530059190711,0.65739547810823,-0.725591006355086],[0,0,0,0],[8.999999E+09,8.999999E+09,8.999999E+09,8.999999E+09,8.999999E+09,8.999999E+09]];
	LOCAL CONST Robtarget Tr_meulage_bavure_P133 :=[[-104.032625,139.779359375,23],[0.146711836765565,-0.132665698517415,0.657457244962017,-0.727066310893797],[0,0,0,0],[8.999999E+09,8.999999E+09,8.999999E+09,8.999999E+09,8.999999E+09,8.999999E+09]];
	LOCAL CONST Robtarget Tr_meulage_bavure_P134 :=[[-103.578125,139.663328125,23],[0.141552725454467,-0.127692913938171,0.657536391467359,-0.728905507965521],[0,0,0,0],[8.999999E+09,8.999999E+09,8.999999E+09,8.999999E+09,8.999999E+09,8.999999E+09]];
	LOCAL CONST Robtarget Tr_meulage_bavure_P135 :=[[-98.273375,140.78409375,23],[0.136041590527842,-0.122379680159976,0.65749809219632,-0.730898185993642],[0,0,0,0],[8.999999E+09,8.999999E+09,8.999999E+09,8.999999E+09,8.999999E+09,8.999999E+09]];
	LOCAL CONST Robtarget Tr_meulage_bavure_P136 :=[[-94.0906640625,142.32440625,23],[0.131295598966521,-0.11775629050818,0.657214001086879,-0.732778737760009],[0,0,0,0],[8.999999E+09,8.999999E+09,8.999999E+09,8.999999E+09,8.999999E+09,8.999999E+09]];
	LOCAL CONST Robtarget Tr_meulage_bavure_P137 :=[[-90.7126171875,142.525,23],[0.128453872875043,-0.114856070161012,0.65657850961029,-0.734310796875888],[0,0,0,0],[8.999999E+09,8.999999E+09,8.999999E+09,8.999999E+09,8.999999E+09,8.999999E+09]];
	LOCAL CONST Robtarget Tr_meulage_bavure_P138 :=[[-86.2345,143.279234375,23],[0.128375461096551,-0.114448230125483,0.655541257319332,-0.735314220970588],[0,0,0,0],[8.999999E+09,8.999999E+09,8.999999E+09,8.999999E+09,8.999999E+09,8.999999E+09]];
	LOCAL CONST Robtarget Tr_meulage_bavure_P139 :=[[-86.203125,143.292453125,23],[0.131580981092875,-0.116996376142597,0.654095430474242,-0.735634053872475],[0,0,0,0],[8.999999E+09,8.999999E+09,8.999999E+09,8.999999E+09,8.999999E+09,8.999999E+09]];
	LOCAL CONST Robtarget Tr_meulage_bavure_P140 :=[[-82.192140625,145.729125,23],[0.138297457892746,-0.122702462497657,0.652231331564391,-0.735127342004878],[0,0,0,0],[8.999999E+09,8.999999E+09,8.999999E+09,8.999999E+09,8.999999E+09,8.999999E+09]];
	LOCAL CONST Robtarget Tr_meulage_bavure_P141 :=[[-78.507078125,145.4126875,23],[0.1484572582451,-0.131512783504132,0.649925237050083,-0.733663421805079],[0,0,0,0],[8.999999E+09,8.999999E+09,8.999999E+09,8.999999E+09,8.999999E+09,8.999999E+09]];
	LOCAL CONST Robtarget Tr_meulage_bavure_P142 :=[[-75.921390625,146.10934375,23],[0.161338708214968,-0.142808737536346,0.647229992944136,-0.731210518215058],[0,0,0,0],[8.999999E+09,8.999999E+09,8.999999E+09,8.999999E+09,8.999999E+09,8.999999E+09]];
	LOCAL CONST Robtarget Tr_meulage_bavure_P143 :=[[-74.7984609375,147.043796875,23],[0.1752245708918,-0.155103321717706,0.644402961248009,-0.728000091265596],[0,0,0,0],[8.999999E+09,8.999999E+09,8.999999E+09,8.999999E+09,8.999999E+09,8.999999E+09]];
	LOCAL CONST Robtarget Tr_meulage_bavure_P144 :=[[-73.9298984375,147.591828125,23],[0.18746458545959,-0.166089545830282,0.642009986535651,-0.724634024285948],[0,0,0,0],[8.999999E+09,8.999999E+09,8.999999E+09,8.999999E+09,8.999999E+09,8.999999E+09]];
	LOCAL CONST Robtarget Tr_meulage_bavure_P145 :=[[-67.570890625,150.951265625,23],[0.195227056615203,-0.173279916080894,0.640802351243267,-0.721964551546309],[0,0,0,0],[8.999999E+09,8.999999E+09,8.999999E+09,8.999999E+09,8.999999E+09,8.999999E+09]];
	LOCAL CONST Robtarget Tr_meulage_bavure_P146 :=[[-66.9260546875,151.566953125,23],[0.19655865752041,-0.174929050846572,0.641383082320086,-0.720688742133022],[0,0,0,0],[8.999999E+09,8.999999E+09,8.999999E+09,8.999999E+09,8.999999E+09,8.999999E+09]];
	LOCAL CONST Robtarget Tr_meulage_bavure_P147 :=[[-64.8245859375,153.340125,23],[0.191130854529928,-0.170690484009002,0.643856728351576,-0.720959269634448],[0,0,0,0],[8.999999E+09,8.999999E+09,8.999999E+09,8.999999E+09,8.999999E+09,8.999999E+09]];
	LOCAL CONST Robtarget Tr_meulage_bavure_P148 :=[[-62.8503125,154.698546875,23],[0.180441545274103,-0.161819445251168,0.64773914327151,-0.722280636699883],[0,0,0,0],[8.999999E+09,8.999999E+09,8.999999E+09,8.999999E+09,8.999999E+09,8.999999E+09]];
	LOCAL CONST Robtarget Tr_meulage_bavure_P149 :=[[-62.48559375,154.97553125,23],[0.16716210886713,-0.150626167439265,0.65224060340869,-0.723844446208383],[0,0,0,0],[8.999999E+09,8.999999E+09,8.999999E+09,8.999999E+09,8.999999E+09,8.999999E+09]];
	LOCAL CONST Robtarget Tr_meulage_bavure_P150 :=[[-59.9157109375,155.998328125,23],[0.154170467926661,-0.139647215122186,0.656650332432079,-0.72494169630718],[0,0,0,0],[8.999999E+09,8.999999E+09,8.999999E+09,8.999999E+09,8.999999E+09,8.999999E+09]];
	LOCAL CONST Robtarget Tr_meulage_bavure_P151 :=[[-58.8825703125,156.425390625,23],[0.143552933911563,-0.130754638205875,0.660566297744076,-0.725222687205604],[0,0,0,0],[8.999999E+09,8.999999E+09,8.999999E+09,8.999999E+09,8.999999E+09,8.999999E+09]];
	LOCAL CONST Robtarget Tr_meulage_bavure_P152 :=[[-56.307375,157.295984375,23],[0.13619474894441,-0.124764748414467,0.663865740427673,-0.724684087447393],[0,0,0,0],[8.999999E+09,8.999999E+09,8.999999E+09,8.999999E+09,8.999999E+09,8.999999E+09]];
	LOCAL CONST Robtarget Tr_meulage_bavure_P153 :=[[-52.86923046875,158.493984375,23],[0.131908539891888,-0.121538788957446,0.666619744827803,-0.723496078557488],[0,0,0,0],[8.999999E+09,8.999999E+09,8.999999E+09,8.999999E+09,8.999999E+09,8.999999E+09]];
	LOCAL CONST Robtarget Tr_meulage_bavure_P154 :=[[-51.7835703125,158.931546875,23],[0.129906182813532,-0.120382215692133,0.668962755296809,-0.721887344284114],[0,0,0,0],[8.999999E+09,8.999999E+09,8.999999E+09,8.999999E+09,8.999999E+09,8.999999E+09]];
	LOCAL CONST Robtarget Tr_meulage_bavure_P155 :=[[-40.98583984375,163.068,23],[0.129305891720435,-0.120495332801063,0.671009997750847,-0.720073915690572],[0,0,0,0],[8.999999E+09,8.999999E+09,8.999999E+09,8.999999E+09,8.999999E+09,8.999999E+09]];
	LOCAL CONST Robtarget Tr_meulage_bavure_P156 :=[[-38.021515625,164.108671875,23],[0.129373227639445,-0.12120583074536,0.67286673639095,-0.718207539379858],[0,0,0,0],[8.999999E+09,8.999999E+09,8.999999E+09,8.999999E+09,8.999999E+09,8.999999E+09]];
	LOCAL CONST Robtarget Tr_meulage_bavure_P157 :=[[-35.14184375,165.060328125,23],[0.129621910662267,-0.122058282314547,0.674593474755252,-0.716396244973632],[0,0,0,0],[8.999999E+09,8.999999E+09,8.999999E+09,8.999999E+09,8.999999E+09,8.999999E+09]];
	LOCAL CONST Robtarget Tr_meulage_bavure_P158 :=[[-33.10540625,165.86828125,23],[0.129759824858608,-0.122773439951585,0.676226762070396,-0.714707238353513],[0,0,0,0],[8.999999E+09,8.999999E+09,8.999999E+09,8.999999E+09,8.999999E+09,8.999999E+09]];
	LOCAL CONST Robtarget Tr_meulage_bavure_P159 :=[[-27.68307421875,168.024234375,23],[0.129668607543797,-0.123239728798151,0.677796862160184,-0.713154566071914],[0,0,0,0],[8.999999E+09,8.999999E+09,8.999999E+09,8.999999E+09,8.999999E+09,8.999999E+09]];
	LOCAL CONST Robtarget Tr_meulage_bavure_P160 :=[[-25.93048046875,168.741875,23],[0.129367059154523,-0.123470253549784,0.679297612590535,-0.711740130962742],[0,0,0,0],[8.999999E+09,8.999999E+09,8.999999E+09,8.999999E+09,8.999999E+09,8.999999E+09]];
	LOCAL CONST Robtarget Tr_meulage_bavure_P161 :=[[-23.64306640625,169.603484375,23],[0.128964069686318,-0.123570265635982,0.680721259328454,-0.710434532718448],[0,0,0,0],[8.999999E+09,8.999999E+09,8.999999E+09,8.999999E+09,8.999999E+09,8.999999E+09]];
	LOCAL CONST Robtarget Tr_meulage_bavure_P162 :=[[-21.365294921875,170.37096875,23],[0.128623608841028,-0.123701790460246,0.682055311303151,-0.709192771119955],[0,0,0,0],[8.999999E+09,8.999999E+09,8.999999E+09,8.999999E+09,8.999999E+09,8.999999E+09]];
	LOCAL CONST Robtarget Tr_meulage_bavure_P163 :=[[-16.819091796875,171.9710625,23],[0.128491255026211,-0.124011131661718,0.683289051568204,-0.707974087529193],[0,0,0,0],[8.999999E+09,8.999999E+09,8.999999E+09,8.999999E+09,8.999999E+09,8.999999E+09]];
	LOCAL CONST Robtarget Tr_meulage_bavure_P164 :=[[-15.8587646484375,172.287046875,23],[0.128632528923293,-0.124566005546947,0.684417153567141,-0.706760314864898],[0,0,0,0],[8.999999E+09,8.999999E+09,8.999999E+09,8.999999E+09,8.999999E+09,8.999999E+09]];
	LOCAL CONST Robtarget Tr_meulage_bavure_P165 :=[[-12.4654541015625,173.585234375,23],[0.129011315999344,-0.125338156547331,0.685457489248446,-0.705545503345213],[0,0,0,0],[8.999999E+09,8.999999E+09,8.999999E+09,8.999999E+09,8.999999E+09,8.999999E+09]];
	LOCAL CONST Robtarget Tr_meulage_bavure_P166 :=[[-5.41607666015625,176.28353125,23],[0.129511301279121,-0.126220599843189,0.686442067516231,-0.704338321377062],[0,0,0,0],[8.999999E+09,8.999999E+09,8.999999E+09,8.999999E+09,8.999999E+09,8.999999E+09]];
	LOCAL CONST Robtarget Tr_meulage_bavure_P167 :=[[-0.180450439453125,178.310421875,23],[0.129996977866521,-0.127085452085077,0.687404886977682,-0.703153322521555],[0,0,0,0],[8.999999E+09,8.999999E+09,8.999999E+09,8.999999E+09,8.999999E+09,8.999999E+09]];
	LOCAL CONST Robtarget Tr_meulage_bavure_P168 :=[[1.27627563476563,178.891109375,23],[0.130370092759055,-0.127835681999483,0.688362923931142,-0.702010087020615],[0,0,0,0],[8.999999E+09,8.999999E+09,8.999999E+09,8.999999E+09,8.999999E+09,8.999999E+09]];
	LOCAL CONST Robtarget Tr_meulage_bavure_P169 :=[[5.4862978515625,180.55865625,23],[0.130586322584719,-0.128427881484974,0.689328343756852,-0.700913636694647],[0,0,0,0],[8.999999E+09,8.999999E+09,8.999999E+09,8.999999E+09,8.999999E+09,8.999999E+09]];
	LOCAL CONST Robtarget Tr_meulage_bavure_P170 :=[[9.74334765625,182.21846875,23],[0.130651814025857,-0.128864426645106,0.690294795460973,-0.699869386669166],[0,0,0,0],[8.999999E+09,8.999999E+09,8.999999E+09,8.999999E+09,8.999999E+09,8.999999E+09]];
	LOCAL CONST Robtarget Tr_meulage_bavure_P171 :=[[15.357849609375,184.33625,23],[0.130576509619386,-0.12915637530599,0.691267764199235,-0.698868574220094],[0,0,0,0],[8.999999E+09,8.999999E+09,8.999999E+09,8.999999E+09,8.999999E+09,8.999999E+09]];
	LOCAL CONST Robtarget Tr_meulage_bavure_P172 :=[[18.40124609375,185.537328125,23],[0.130334806168128,-0.129274589622324,0.692245807004908,-0.697923105695191],[0,0,0,0],[8.999999E+09,8.999999E+09,8.999999E+09,8.999999E+09,8.999999E+09,8.999999E+09]];
	LOCAL CONST Robtarget Tr_meulage_bavure_P173 :=[[22.57159375,187.19659375,23],[0.129865960091058,-0.12915605292908,0.6932373426365,-0.697047726612527],[0,0,0,0],[8.999999E+09,8.999999E+09,8.999999E+09,8.999999E+09,8.999999E+09,8.999999E+09]];
	LOCAL CONST Robtarget Tr_meulage_bavure_P174 :=[[22.874939453125,187.317625,23],[0.129131800597102,-0.128759034957762,0.694244678975425,-0.6962545617126],[0,0,0,0],[8.999999E+09,8.999999E+09,8.999999E+09,8.999999E+09,8.999999E+09,8.999999E+09]];
	LOCAL CONST Robtarget Tr_meulage_bavure_P175 :=[[23.29376171875,187.488734375,23],[0.128181521688233,-0.128130089501948,0.69525679964137,-0.695535879889997],[0,0,0,0],[8.999999E+09,8.999999E+09,8.999999E+09,8.999999E+09,8.999999E+09,8.999999E+09]];
	LOCAL CONST Robtarget Tr_meulage_bavure_P176 :=[[32.046173828125,191.0809375,23],[0.127187591411657,-0.127438697195851,0.696236706397722,-0.694864838448729],[0,0,0,0],[8.999999E+09,8.999999E+09,8.999999E+09,8.999999E+09,8.999999E+09,8.999999E+09]];
	LOCAL CONST Robtarget Tr_meulage_bavure_P177 :=[[37.37878515625,193.0600625,23],[0.126419470687451,-0.126954897011015,0.697133866170125,-0.694193736787304],[0,0,0,0],[8.999999E+09,8.999999E+09,8.999999E+09,8.999999E+09,8.999999E+09,8.999999E+09]];
	LOCAL CONST Robtarget Tr_meulage_bavure_P178 :=[[37.698578125,193.17725,23],[0.126117548604661,-0.126921776395056,0.697903361883251,-0.693481163466413],[0,0,0,0],[8.999999E+09,8.999999E+09,8.999999E+09,8.999999E+09,8.999999E+09,8.999999E+09]];
	LOCAL CONST Robtarget Tr_meulage_bavure_P179 :=[[40.8884296875,194.392734375,23],[0.126380009559147,-0.127441690503163,0.69852796991901,-0.692708729515048],[0,0,0,0],[8.999999E+09,8.999999E+09,8.999999E+09,8.999999E+09,8.999999E+09,8.999999E+09]];
	LOCAL CONST Robtarget Tr_meulage_bavure_P180 :=[[45.28210546875,196.084015625,23],[0.127058885510676,-0.1283676349692,0.699031756369221,-0.691904902058484],[0,0,0,0],[8.999999E+09,8.999999E+09,8.999999E+09,8.999999E+09,8.999999E+09,8.999999E+09]];
	LOCAL CONST Robtarget Tr_meulage_bavure_P181 :=[[49.8389296875,197.72396875,23],[0.127597082891395,-0.129136744629311,0.699514544783177,-0.6911744260756],[0,0,0,0],[8.999999E+09,8.999999E+09,8.999999E+09,8.999999E+09,8.999999E+09,8.999999E+09]];
	LOCAL CONST Robtarget Tr_meulage_bavure_P182 :=[[58.59753515625,201.009453125,23],[0.127042256256765,-0.128785526320427,0.700162984312058,-0.690685419518028],[0,0,0,0],[8.999999E+09,8.999999E+09,8.999999E+09,8.999999E+09,8.999999E+09,8.999999E+09]];
	LOCAL CONST Robtarget Tr_meulage_bavure_P183 :=[[60.100890625,201.62865625,23],[0.123936934519371,-0.125829763227576,0.701245194294732,-0.690696521220845],[0,0,0,0],[8.999999E+09,8.999999E+09,8.999999E+09,8.999999E+09,8.999999E+09,8.999999E+09]];
	LOCAL CONST Robtarget Tr_meulage_bavure_P184 :=[[62.44671484375,202.59871875,23],[0.116286282002992,-0.118229192334943,0.703069039764045,-0.691515208815404],[0,0,0,0],[8.999999E+09,8.999999E+09,8.999999E+09,8.999999E+09,8.999999E+09,8.999999E+09]];
	LOCAL CONST Robtarget Tr_meulage_bavure_P185 :=[[64.86050390625,203.50121875,23],[0.101683369222815,-0.103518518715243,0.705851501688481,-0.693338349055217],[0,0,0,0],[8.999999E+09,8.999999E+09,8.999999E+09,8.999999E+09,8.999999E+09,8.999999E+09]];
	LOCAL CONST Robtarget Tr_meulage_bavure_P186 :=[[68.275875,204.921234375,23],[0.0775958802939646,-0.0790938314470255,0.709438705096916,-0.696002707537008],[0,0,0,0],[8.999999E+09,8.999999E+09,8.999999E+09,8.999999E+09,8.999999E+09,8.999999E+09]];
	LOCAL CONST Robtarget Tr_meulage_bavure_P187 :=[[71.1980859375,206.141171875,23],[0.0418939640137601,-0.042750962084207,0.712948765151269,-0.698656789338921],[0,0,0,0],[8.999999E+09,8.999999E+09,8.999999E+09,8.999999E+09,8.999999E+09,8.999999E+09]];
	LOCAL CONST Robtarget Tr_meulage_bavure_P188 :=[[72.951328125,206.808015625,23],[0.00650736295723059,-0.00664740229093401,-0.714562892303787,0.699509356057924],[0,0,0,0],[8.999999E+09,8.999999E+09,8.999999E+09,8.999999E+09,8.999999E+09,8.999999E+09]];
	LOCAL CONST Robtarget Tr_meulage_bavure_P189 :=[[75.2215,207.202640625,23],[0.0668250541541537,-0.0683287659253594,-0.711657032158465,0.695995589399687],[0,0,0,0],[8.999999E+09,8.999999E+09,8.999999E+09,8.999999E+09,8.999999E+09,8.999999E+09]];
	LOCAL CONST Robtarget Tr_meulage_bavure_P190 :=[[77.3096640625,207.633734375,23],[0.135946770846249,-0.139127314222613,-0.701572905816659,0.685534480356495],[0,0,0,0],[8.999999E+09,8.999999E+09,8.999999E+09,8.999999E+09,8.999999E+09,8.999999E+09]];
	LOCAL CONST Robtarget Tr_meulage_bavure_P191 :=[[79.4188203125,206.551265625,23],[0.208490173434681,-0.213535310755655,-0.682902293622158,0.666767557704526],[0,0,0,0],[8.999999E+09,8.999999E+09,8.999999E+09,8.999999E+09,8.999999E+09,8.999999E+09]];
	LOCAL CONST Robtarget Tr_meulage_bavure_P192 :=[[80.0400703125,206.331109375,23],[0.277730766130165,-0.284646817401559,-0.65671318576587,0.640757054217241],[0,0,0,0],[8.999999E+09,8.999999E+09,8.999999E+09,8.999999E+09,8.999999E+09,8.999999E+09]];
	LOCAL CONST Robtarget Tr_meulage_bavure_P193 :=[[81.567015625,203.339421875,23],[0.337441236722282,-0.346050838073459,-0.626772135205383,0.611178304390853],[0,0,0,0],[8.999999E+09,8.999999E+09,8.999999E+09,8.999999E+09,8.999999E+09,8.999999E+09]];
	LOCAL CONST Robtarget Tr_meulage_bavure_P194 :=[[81.8603828125,202.80884375,23],[0.384088930902801,-0.394090741726273,-0.597949156809868,0.582773529180887],[0,0,0,0],[8.999999E+09,8.999999E+09,8.999999E+09,8.999999E+09,8.999999E+09,8.999999E+09]];
	LOCAL CONST Robtarget Tr_meulage_bavure_P195 :=[[81.8648359375,202.806765625,23],[0.417485445412743,-0.428533535492199,-0.573947469263428,0.559150439822045],[0,0,0,0],[8.999999E+09,8.999999E+09,8.999999E+09,8.999999E+09,8.999999E+09,8.999999E+09]];
	LOCAL CONST Robtarget Tr_meulage_bavure_P196 :=[[81.9259375,202.649359375,23],[0.439669980581897,-0.451452642152384,-0.556246769008926,0.541729039313821],[0,0,0,0],[8.999999E+09,8.999999E+09,8.999999E+09,8.999999E+09,8.999999E+09,8.999999E+09]];
	LOCAL CONST Robtarget Tr_meulage_bavure_P197 :=[[81.9753125,202.195125,23],[0.453411471570483,-0.465669511787846,-0.544506027073574,0.530172735738184],[0,0,0,0],[8.999999E+09,8.999999E+09,8.999999E+09,8.999999E+09,8.999999E+09,8.999999E+09]];
	LOCAL CONST Robtarget Tr_meulage_bavure_P198 :=[[82.1716953125,200.726875,23],[0.461363787734214,-0.473901876204428,-0.537420239762482,0.523201637030217],[0,0,0,0],[8.999999E+09,8.999999E+09,8.999999E+09,8.999999E+09,8.999999E+09,8.999999E+09]];
	LOCAL CONST Robtarget Tr_meulage_bavure_P199 :=[[82.2009609375,200.3215,23],[0.465648460503174,-0.478321715727243,-0.533508574901795,0.519373129841183],[0,0,0,0],[8.999999E+09,8.999999E+09,8.999999E+09,8.999999E+09,8.999999E+09,8.999999E+09]];
	LOCAL CONST Robtarget Tr_meulage_bavure_P200 :=[[82.60821875,195.031796875,23],[0.467782316371388,-0.480479987086091,-0.531532730755952,0.517485886411494],[0,0,0,0],[8.999999E+09,8.999999E+09,8.999999E+09,8.999999E+09,8.999999E+09,8.999999E+09]];
	LOCAL CONST Robtarget Tr_meulage_bavure_P201 :=[[83.064609375,189.71584375,23],[0.468714650503222,-0.481355775818431,-0.53065970573775,0.516723785204632],[0,0,0,0],[8.999999E+09,8.999999E+09,8.999999E+09,8.999999E+09,8.999999E+09,8.999999E+09]];
	LOCAL CONST Robtarget Tr_meulage_bavure_P202 :=[[83.291078125,186.89309375,23],[0.468844012391605,-0.481353271614545,-0.530529597660492,0.516742359359779],[0,0,0,0],[8.999999E+09,8.999999E+09,8.999999E+09,8.999999E+09,8.999999E+09,8.999999E+09]];
	LOCAL CONST Robtarget Tr_meulage_bavure_P203 :=[[83.4083828125,185.326875,23],[0.468180954746477,-0.480476112195577,-0.531131924445055,0.517540508614923],[0,0,0,0],[8.999999E+09,8.999999E+09,8.999999E+09,8.999999E+09,8.999999E+09,8.999999E+09]];
	LOCAL CONST Robtarget Tr_meulage_bavure_P204 :=[[83.80996875,181.384953125,23],[0.466317227457552,-0.478311603410114,-0.532835257604839,0.519473619804444],[0,0,0,0],[8.999999E+09,8.999999E+09,8.999999E+09,8.999999E+09,8.999999E+09,8.999999E+09]];
	LOCAL CONST Robtarget Tr_meulage_bavure_P205 :=[[84.4078046875,176.141171875,23],[0.462507536012093,-0.474093594474114,-0.536286951131274,0.523180990534785],[0,0,0,0],[8.999999E+09,8.999999E+09,8.999999E+09,8.999999E+09,8.999999E+09,8.999999E+09]];
	LOCAL CONST Robtarget Tr_meulage_bavure_P206 :=[[84.74215625,173.671625,23],[0.456035160102432,-0.467093778601475,-0.542034296031581,0.529201432979631],[0,0,0,0],[8.999999E+09,8.999999E+09,8.999999E+09,8.999999E+09,8.999999E+09,8.999999E+09]];
	LOCAL CONST Robtarget Tr_meulage_bavure_P207 :=[[84.9359453125,171.51334375,23],[0.446739713010516,-0.457153573794796,-0.550027452426193,0.537497944520237],[0,0,0,0],[8.999999E+09,8.999999E+09,8.999999E+09,8.999999E+09,8.999999E+09,8.999999E+09]];
	LOCAL CONST Robtarget Tr_meulage_bavure_P208 :=[[84.9572109375,170.9715,23],[0.435678808601492,-0.445372563430718,-0.559146164584857,0.546976070874019],[0,0,0,0],[8.999999E+09,8.999999E+09,8.999999E+09,8.999999E+09,8.999999E+09,8.999999E+09]];
	LOCAL CONST Robtarget Tr_meulage_bavure_P209 :=[[85.00009375,170.01140625,23],[0.425397514108343,-0.434360413506672,-0.567234350844906,0.555529636824457],[0,0,0,0],[8.999999E+09,8.999999E+09,8.999999E+09,8.999999E+09,8.999999E+09,8.999999E+09]];
	LOCAL CONST Robtarget Tr_meulage_bavure_P210 :=[[85.3654140625,161.88396875,23],[0.419210597935592,-0.427495246625982,-0.571866630278364,0.560784134819044],[0,0,0,0],[8.999999E+09,8.999999E+09,8.999999E+09,8.999999E+09,8.999999E+09,8.999999E+09]];
	LOCAL CONST Robtarget Tr_meulage_bavure_P211 :=[[85.462375,161.8231875,23],[0.419579838624585,-0.427286389263082,-0.571424245439722,0.561118019933356],[0,0,0,0],[8.999999E+09,8.999999E+09,8.999999E+09,8.999999E+09,8.999999E+09,8.999999E+09]];
	LOCAL CONST Robtarget Tr_meulage_bavure_P212 :=[[85.6098359375,158.448890625,23],[0.426600498102056,-0.43381020671801,-0.56585112588199,0.556446963244871],[0,0,0,0],[8.999999E+09,8.999999E+09,8.999999E+09,8.999999E+09,8.999999E+09,8.999999E+09]];
	LOCAL CONST Robtarget Tr_meulage_bavure_P213 :=[[85.780546875,155.384640625,23],[0.437941124152104,-0.44467437369272,-0.556680342328477,0.548251100885741],[0,0,0,0],[8.999999E+09,8.999999E+09,8.999999E+09,8.999999E+09,8.999999E+09,8.999999E+09]];
	LOCAL CONST Robtarget Tr_meulage_bavure_P214 :=[[86.0823984375,149.711453125,23],[0.450325026944704,-0.456550424145864,-0.54628385742044,0.538834879570103],[0,0,0,0],[8.999999E+09,8.999999E+09,8.999999E+09,8.999999E+09,8.999999E+09,8.999999E+09]];
	LOCAL CONST Robtarget Tr_meulage_bavure_P215 :=[[86.138578125,148.8935,23],[0.461166065904665,-0.466824209471746,-0.536816665304467,0.530310178066088],[0,0,0,0],[8.999999E+09,8.999999E+09,8.999999E+09,8.999999E+09,8.999999E+09,8.999999E+09]];
	LOCAL CONST Robtarget Tr_meulage_bavure_P216 :=[[86.470546875,142.730015625,23],[0.469336260131283,-0.474381314657693,-0.529441358737364,0.523810739569124],[0,0,0,0],[8.999999E+09,8.999999E+09,8.999999E+09,8.999999E+09,8.999999E+09,8.999999E+09]];
	LOCAL CONST Robtarget Tr_meulage_bavure_P217 :=[[86.5939921875,140.929625,23],[0.474947639812807,-0.479356911104891,-0.524249230622284,0.51942702606253],[0,0,0,0],[8.999999E+09,8.999999E+09,8.999999E+09,8.999999E+09,8.999999E+09,8.999999E+09]];
	LOCAL CONST Robtarget Tr_meulage_bavure_P218 :=[[86.7443515625,139.27765625,23],[0.478682510695159,-0.482457094188465,-0.520732452970152,0.516658415827605],[0,0,0,0],[8.999999E+09,8.999999E+09,8.999999E+09,8.999999E+09,8.999999E+09,8.999999E+09]];
	LOCAL CONST Robtarget Tr_meulage_bavure_P219 :=[[86.8099375,137.8385,23],[0.481244849432884,-0.484412560449389,-0.518290269353855,0.514901022397797],[0,0,0,0],[8.999999E+09,8.999999E+09,8.999999E+09,8.999999E+09,8.999999E+09,8.999999E+09]];
	LOCAL CONST Robtarget Tr_meulage_bavure_P220 :=[[86.8993203125,135.272765625,23],[0.483033791313791,-0.485627612176269,-0.516569008445365,0.513809924247062],[0,0,0,0],[8.999999E+09,8.999999E+09,8.999999E+09,8.999999E+09,8.999999E+09,8.999999E+09]];
	LOCAL CONST Robtarget Tr_meulage_bavure_P221 :=[[86.9025859375,134.49471875,23],[0.484243066107561,-0.486309726462873,-0.515395192523988,0.513204928266978],[0,0,0,0],[8.999999E+09,8.999999E+09,8.999999E+09,8.999999E+09,8.999999E+09,8.999999E+09]];
	LOCAL CONST Robtarget Tr_meulage_bavure_P222 :=[[86.9266953125,132.059484375,23],[0.485002451720835,-0.48658745139277,-0.514649389571461,0.512972981535665],[0,0,0,0],[8.999999E+09,8.999999E+09,8.999999E+09,8.999999E+09,8.999999E+09,8.999999E+09]];
	LOCAL CONST Robtarget Tr_meulage_bavure_P223 :=[[86.9136328125,130.817109375,23],[0.485427827166442,-0.486569890302561,-0.514222427614951,0.513015459222436],[0,0,0,0],[8.999999E+09,8.999999E+09,8.999999E+09,8.999999E+09,8.999999E+09,8.999999E+09]];
	LOCAL CONST Robtarget Tr_meulage_bavure_P224 :=[[86.975953125,129.6813359375,23],[0.485716023054186,-0.486456158277755,-0.513927744690145,0.513145811889539],[0,0,0,0],[8.999999E+09,8.999999E+09,8.999999E+09,8.999999E+09,8.999999E+09,8.999999E+09]];
	LOCAL CONST Robtarget Tr_meulage_bavure_P225 :=[[87.2295859375,125.4028046875,23],[0.486067155951361,-0.486430682860973,-0.513574724982401,0.513190912366942],[0,0,0,0],[8.999999E+09,8.999999E+09,8.999999E+09,8.999999E+09,8.999999E+09,8.999999E+09]];
	LOCAL CONST Robtarget Tr_meulage_bavure_P226 :=[[87.3719140625,122.88946875,23],[0.486579063055982,-0.486582382488066,-0.513070166770623,0.513066666640667],[0,0,0,0],[8.999999E+09,8.999999E+09,8.999999E+09,8.999999E+09,8.999999E+09,8.999999E+09]];
	LOCAL CONST Robtarget Tr_meulage_bavure_P227 :=[[87.5888671875,120.5894453125,23],[0.487234613660268,-0.486884506362452,-0.51242957407672,0.512798050237198],[0,0,0,0],[8.999999E+09,8.999999E+09,8.999999E+09,8.999999E+09,8.999999E+09,8.999999E+09]];
	LOCAL CONST Robtarget Tr_meulage_bavure_P228 :=[[87.7881484375,117.7775859375,23],[0.487923074783589,-0.487206417931878,-0.511756750481601,0.512509519673761],[0,0,0,0],[8.999999E+09,8.999999E+09,8.999999E+09,8.999999E+09,8.999999E+09,8.999999E+09]];
	LOCAL CONST Robtarget Tr_meulage_bavure_P229 :=[[88.0114140625,112.2958359375,23],[0.488488070136954,-0.487386990594344,-0.511200179119025,0.512355056188518],[0,0,0,0],[8.999999E+09,8.999999E+09,8.999999E+09,8.999999E+09,8.999999E+09,8.999999E+09]];
	LOCAL CONST Robtarget Tr_meulage_bavure_P230 :=[[88.210234375,107.0625,23],[0.488804684781886,-0.487290344885852,-0.510878358134093,0.512466001903075],[0,0,0,0],[8.999999E+09,8.999999E+09,8.999999E+09,8.999999E+09,8.999999E+09,8.999999E+09]];
	LOCAL CONST Robtarget Tr_meulage_bavure_P231 :=[[88.36725,103.8018515625,23],[0.48880864858073,-0.486842909056306,-0.510851439652514,0.512914119106921],[0,0,0,0],[8.999999E+09,8.999999E+09,8.999999E+09,8.999999E+09,8.999999E+09,8.999999E+09]];
	LOCAL CONST Robtarget Tr_meulage_bavure_P232 :=[[88.4679296875,101.3322734375,23],[0.488515615429702,-0.486055438334638,-0.511102492470296,0.513689445616039],[0,0,0,0],[8.999999E+09,8.999999E+09,8.999999E+09,8.999999E+09,8.999999E+09,8.999999E+09]];
	LOCAL CONST Robtarget Tr_meulage_bavure_P233 :=[[88.4963046875,99.366546875,23],[0.488016790478025,-0.485012840355096,-0.511542139716795,0.514710400318638],[0,0,0,0],[8.999999E+09,8.999999E+09,8.999999E+09,8.999999E+09,8.999999E+09,8.999999E+09]];
	LOCAL CONST Robtarget Tr_meulage_bavure_P234 :=[[88.8017890625,96.0728125,23],[0.487447564676569,-0.483859404695169,-0.512040985051918,0.515838131399744],[0,0,0,0],[8.999999E+09,8.999999E+09,8.999999E+09,8.999999E+09,8.999999E+09,8.999999E+09]];
	LOCAL CONST Robtarget Tr_meulage_bavure_P235 :=[[88.92840625,93.9544375,23],[0.486972688480907,-0.482750693068154,-0.512443203376377,0.516924880741149],[0,0,0,0],[8.999999E+09,8.999999E+09,8.999999E+09,8.999999E+09,8.999999E+09,8.999999E+09]];
	LOCAL CONST Robtarget Tr_meulage_bavure_P236 :=[[89.0796484375,92.279390625,23],[0.486736129209475,-0.481830496072847,-0.512615513700911,0.517834576568157],[0,0,0,0],[8.999999E+09,8.999999E+09,8.999999E+09,8.999999E+09,8.999999E+09,8.999999E+09]];
	LOCAL CONST Robtarget Tr_meulage_bavure_P237 :=[[89.1046171875,91.3662734375,23],[0.486820548476699,-0.481195030834756,-0.512484289437609,0.518475601123536],[0,0,0,0],[8.999999E+09,8.999999E+09,8.999999E+09,8.999999E+09,8.999999E+09,8.999999E+09]];
	LOCAL CONST Robtarget Tr_meulage_bavure_P238 :=[[89.1337578125,90.875515625,23],[0.487232102641729,-0.480848079756631,-0.512045791157769,0.518844013271131],[0,0,0,0],[8.999999E+09,8.999999E+09,8.999999E+09,8.999999E+09,8.999999E+09,8.999999E+09]];
	LOCAL CONST Robtarget Tr_meulage_bavure_P239 :=[[89.16028125,89.797359375,23],[0.487896548066862,-0.480722305305391,-0.511370510333837,0.519002143278062],[0,0,0,0],[8.999999E+09,8.999999E+09,8.999999E+09,8.999999E+09,8.999999E+09,8.999999E+09]];
	LOCAL CONST Robtarget Tr_meulage_bavure_P240 :=[[89.189546875,88.7360546875,23],[0.488682597852706,-0.480701598802967,-0.510581501930545,0.519058591442768],[0,0,0,0],[8.999999E+09,8.999999E+09,8.999999E+09,8.999999E+09,8.999999E+09,8.999999E+09]];
	LOCAL CONST Robtarget Tr_meulage_bavure_P241 :=[[89.5481875,80.2841171875,23],[0.489462179395491,-0.480667394360316,-0.509798022047976,0.519125811009481],[0,0,0,0],[8.999999E+09,8.999999E+09,8.999999E+09,8.999999E+09,8.999999E+09,8.999999E+09]];
	LOCAL CONST Robtarget Tr_meulage_bavure_P242 :=[[89.623140625,79.6325390625,23],[0.490141303111174,-0.480541214545683,-0.509108111086435,0.519278899372431],[0,0,0,0],[8.999999E+09,8.999999E+09,8.999999E+09,8.999999E+09,8.999999E+09,8.999999E+09]];
	LOCAL CONST Robtarget Tr_meulage_bavure_P243 :=[[89.6957421875,78.3010859375,23],[0.490696201435401,-0.480306316336964,-0.508534074142616,0.519534576154076],[0,0,0,0],[8.999999E+09,8.999999E+09,8.999999E+09,8.999999E+09,8.999999E+09,8.999999E+09]];
	LOCAL CONST Robtarget Tr_meulage_bavure_P244 :=[[89.6254609375,77.276578125,23],[0.491163699481001,-0.480021511004312,-0.5080433887249,0.519836016892053],[0,0,0,0],[8.999999E+09,8.999999E+09,8.999999E+09,8.999999E+09,8.999999E+09,8.999999E+09]];
	LOCAL CONST Robtarget Tr_meulage_bavure_P245 :=[[89.64715625,76.986359375,23],[0.491615604671525,-0.479770251518427,-0.507570720875201,0.520102457513542],[0,0,0,0],[8.999999E+09,8.999999E+09,8.999999E+09,8.999999E+09,8.999999E+09,8.999999E+09]];
	LOCAL CONST Robtarget Tr_meulage_bavure_P246 :=[[89.7738671875,75.3290703125,23],[0.492139312926278,-0.4796389462415,-0.507035714032184,0.520250096219758],[0,0,0,0],[8.999999E+09,8.999999E+09,8.999999E+09,8.999999E+09,8.999999E+09,8.999999E+09]];
	LOCAL CONST Robtarget Tr_meulage_bavure_P247 :=[[90.246125,69.478640625,23],[0.492797044477793,-0.479709062869272,-0.506382916162728,0.520198644917082],[0,0,0,0],[8.999999E+09,8.999999E+09,8.999999E+09,8.999999E+09,8.999999E+09,8.999999E+09]];
	LOCAL CONST Robtarget Tr_meulage_bavure_P248 :=[[90.38025,67.148953125,23],[0.493609551655298,-0.480012163578399,-0.505593972252053,0.519916020674331],[0,0,0,0],[8.999999E+09,8.999999E+09,8.999999E+09,8.999999E+09,8.999999E+09,8.999999E+09]];
	LOCAL CONST Robtarget Tr_meulage_bavure_P249 :=[[90.570921875,58.42654296875,23],[0.494545381501658,-0.480520074074132,-0.504697403176773,0.519428392825991],[0,0,0,0],[8.999999E+09,8.999999E+09,8.999999E+09,8.999999E+09,8.999999E+09,8.999999E+09]];
	LOCAL CONST Robtarget Tr_meulage_bavure_P250 :=[[90.6774609375,54.2451171875,23],[0.495491929720599,-0.481131232861917,-0.503797057667085,0.518834278968263],[0,0,0,0],[8.999999E+09,8.999999E+09,8.999999E+09,8.999999E+09,8.999999E+09,8.999999E+09]];
	LOCAL CONST Robtarget Tr_meulage_bavure_P251 :=[[90.73190625,52.53121875,23],[0.496241547391399,-0.481648161062708,-0.503085505526553,0.518328418781562],[0,0,0,0],[8.999999E+09,8.999999E+09,8.999999E+09,8.999999E+09,8.999999E+09,8.999999E+09]];
	LOCAL CONST Robtarget Tr_meulage_bavure_P252 :=[[91.2394375,46.3190625,23],[0.496525673675689,-0.481814579253206,-0.502813407645297,0.518165652752171],[0,0,0,0],[8.999999E+09,8.999999E+09,8.999999E+09,8.999999E+09,8.999999E+09,8.999999E+09]];
	LOCAL CONST Robtarget Tr_meulage_bavure_P253 :=[[91.37384375,44.75738671875,23],[0.496106823281242,-0.481396906449671,-0.503201723616101,0.518577924428206],[0,0,0,0],[8.999999E+09,8.999999E+09,8.999999E+09,8.999999E+09,8.999999E+09,8.999999E+09]];
	LOCAL CONST Robtarget Tr_meulage_bavure_P254 :=[[91.413515625,44.36984375,23],[0.494877687390771,-0.480287784712952,-0.504346635359727,0.519667383794297],[0,0,0,0],[8.999999E+09,8.999999E+09,8.999999E+09,8.999999E+09,8.999999E+09,8.999999E+09]];
	LOCAL CONST Robtarget Tr_meulage_bavure_P255 :=[[91.416046875,44.01062109375,23],[0.492919162077556,-0.478557577322578,-0.50616462143842,0.521354697732749],[0,0,0,0],[8.999999E+09,8.999999E+09,8.999999E+09,8.999999E+09,8.999999E+09,8.999999E+09]];
	LOCAL CONST Robtarget Tr_meulage_bavure_P256 :=[[92.0011015625,39.38336328125,23],[0.490499427326038,-0.476459565226207,-0.508399192178365,0.523380221148705],[0,0,0,0],[8.999999E+09,8.999999E+09,8.999999E+09,8.999999E+09,8.999999E+09,8.999999E+09]];
	LOCAL CONST Robtarget Tr_meulage_bavure_P257 :=[[92.1544765625,37.63262890625,23],[0.487973381874229,-0.474328389817663,-0.510720954676969,0.525412850669886],[0,0,0,0],[8.999999E+09,8.999999E+09,8.999999E+09,8.999999E+09,8.999999E+09,8.999999E+09]];
	LOCAL CONST Robtarget Tr_meulage_bavure_P258 :=[[92.331265625,33.3674609375,23],[0.48569006198071,-0.472492020387984,-0.512815619924968,0.527140013965764],[0,0,0,0],[8.999999E+09,8.999999E+09,8.999999E+09,8.999999E+09,8.999999E+09,8.999999E+09]];
	LOCAL CONST Robtarget Tr_meulage_bavure_P259 :=[[92.607484375,28.623748046875,23],[0.483927868430405,-0.471209979071303,-0.514439769328583,0.528324424490465],[0,0,0,0],[8.999999E+09,8.999999E+09,8.999999E+09,8.999999E+09,8.999999E+09,8.999999E+09]];
	LOCAL CONST Robtarget Tr_meulage_bavure_P260 :=[[92.7828984375,27.233337890625,23],[0.482855043973076,-0.47064188022674,-0.515450782105311,0.528826737517517],[0,0,0,0],[8.999999E+09,8.999999E+09,8.999999E+09,8.999999E+09,8.999999E+09,8.999999E+09]];
	LOCAL CONST Robtarget Tr_meulage_bavure_P261 :=[[93.132265625,24.560546875,23],[0.482525659054035,-0.470832059121889,-0.515803564345592,0.528614078005774],[0,0,0,0],[8.999999E+09,8.999999E+09,8.999999E+09,8.999999E+09,8.999999E+09,8.999999E+09]];
	LOCAL CONST Robtarget Tr_meulage_bavure_P262 :=[[93.2118203125,23.02780078125,23],[0.482848023675962,-0.471685072250217,-0.515577462530979,0.527779176151013],[0,0,0,0],[8.999999E+09,8.999999E+09,8.999999E+09,8.999999E+09,8.999999E+09,8.999999E+09]];
	LOCAL CONST Robtarget Tr_meulage_bavure_P263 :=[[93.2736484375,22.18475390625,23],[0.48357070427211,-0.472952768250357,-0.514991744893841,0.526553468951916],[0,0,0,0],[8.999999E+09,8.999999E+09,8.999999E+09,8.999999E+09,8.999999E+09,8.999999E+09]];
	LOCAL CONST Robtarget Tr_meulage_bavure_P264 :=[[93.2137109375,18.0667109375,23],[0.484324151629945,-0.474270334232257,-0.514374106862114,0.525278063890888],[0,0,0,0],[8.999999E+09,8.999999E+09,8.999999E+09,8.999999E+09,8.999999E+09,8.999999E+09]];
	LOCAL CONST Robtarget Tr_meulage_bavure_P265 :=[[93.168484375,14.9177548828125,23],[0.484717083946662,-0.47525008159203,-0.514078321735536,0.524318784327425],[0,0,0,0],[8.999999E+09,8.999999E+09,8.999999E+09,8.999999E+09,8.999999E+09,8.999999E+09]];
	LOCAL CONST Robtarget Tr_meulage_bavure_P266 :=[[93.4845859375,10.84423828125,23],[0.484439508676399,-0.47558187793763,-0.514389122750501,0.523969531754143],[0,0,0,0],[8.999999E+09,8.999999E+09,8.999999E+09,8.999999E+09,8.999999E+09,8.999999E+09]];
	LOCAL CONST Robtarget Tr_meulage_bavure_P267 :=[[93.6888125,8.7680361328125,23],[0.483344314637207,-0.475121621207879,-0.515442588118126,0.524363096453949],[0,0,0,0],[8.999999E+09,8.999999E+09,8.999999E+09,8.999999E+09,8.999999E+09,8.999999E+09]];
	LOCAL CONST Robtarget Tr_meulage_bavure_P268 :=[[93.7647734375,6.1404111328125,23],[0.481439712260312,-0.473874068070304,-0.517227537803136,0.52548534252376],[0,0,0,0],[8.999999E+09,8.999999E+09,8.999999E+09,8.999999E+09,8.999999E+09,8.999999E+09]];
	LOCAL CONST Robtarget Tr_meulage_bavure_P269 :=[[93.9436328125,2.99270629882813,23],[0.478838013374533,-0.471945714854551,-0.519633094005383,0.527221819343955],[0,0,0,0],[8.999999E+09,8.999999E+09,8.999999E+09,8.999999E+09,8.999999E+09,8.999999E+09]];
